		//Wait for Delay, copy Data and then next step
		IF NOT fbMBRead_FC3.bBusy AND NOT fbMBRead_FC3.bError AND timer_Delay.Q THEN
			m_Poll_ok:=TRUE;
			int_Data_Received:=int_Data_Received+1;
			m_MBTCPError := FALSE; 
			
			FOR i:=0 TO 9 BY 1 DO
				arrBuffer_Received[i + WORD_TO_INT(w_Adress)] := arrBuffer_FC3[i];
			END_FOR
			
			//Go to Next Step
			timer_Timeout.IN := FALSE;
			fbMBRead_FC3.bExecute := FALSE;
			timer_Delay.IN := FALSE;		
			iStateModbusRead := iStateModbusRead+1;
		END_IF	

		//Error or Timeout
		IF FPError_FC_3.Q THEN 
			iStateModbusError := 300;
			int_FC4Error := int_FC4Error+1;
		ELSIF timer_Timeout.Q THEN  
			timer_Timeout.IN := FALSE; 	
			iStateModbusError := 300;
			int_TimeoutError := int_TimeoutError+1;
		END_IF
	
	9://Wait and go to next step
		timer_Wait.IN := TRUE;
		
		IF timer_Wait.Q = TRUE THEN
			iStateModbusRead := iStateModbusRead+1;
			timer_Wait.IN :=FALSE;
		END_IF
		
	10: // clean the array  Poll 4
		FOR i:=0 TO 10 BY 1 DO
			arrBuffer_FC3[i] := 0;
		END_FOR
		w_Adress := w_Adress + 10;
		usint_Quantity := 10; 
		iStateModbusRead := iStateModbusRead+1;
		
	11://read the required registers
		//Start Read Poll 4
		fbMBRead_FC3.nQuantity := usint_Quantity;
		fbMBRead_FC3.nMBAddr := w_Adress;
		fbMBRead_FC3.bExecute := TRUE;
		fbMBRead_FC3.nUnitID := 1;
		timer_Timeout.IN := TRUE;
		IF fbMBRead_FC3.bBusy THEN 
			timer_Delay.IN := TRUE; 
		END_IF
		
		//Wait for Delay, copy Data and then next step
		IF NOT fbMBRead_FC3.bBusy AND NOT fbMBRead_FC3.bError AND timer_Delay.Q THEN
			m_Poll_ok:=TRUE;
			int_Data_Received:=int_Data_Received+1;
			m_MBTCPError := FALSE; 
			
			FOR i:=0 TO 9 BY 1 DO
				arrBuffer_Received[i + WORD_TO_INT(w_Adress)] := arrBuffer_FC3[i];
			END_FOR
			
			//Go to Next Step
			timer_Timeout.IN := FALSE;
			fbMBRead_FC3.bExecute := FALSE;
			timer_Delay.IN := FALSE;		
			iStateModbusRead := iStateModbusRead+1;
		END_IF	

		//Error or Timeout
		IF FPError_FC_3.Q THEN 
			iStateModbusError := 300;
			int_FC4Error := int_FC4Error+1;
		ELSIF timer_Timeout.Q THEN  
			timer_Timeout.IN := FALSE; 	
			iStateModbusError := 300;
			int_TimeoutError := int_TimeoutError+1;
		END_IF
	
	12://Wait and go to next step
		timer_Wait.IN := TRUE;
		
		IF timer_Wait.Q = TRUE THEN
			iStateModbusRead := iStateModbusRead+1;
			timer_Wait.IN :=FALSE;
		END_IF		
		
	13: // clean the array  Poll 4
		FOR i:=0 TO 10 BY 1 DO
			arrBuffer_FC3[i] := 0;
		END_FOR
		w_Adress := w_Adress + 10;
		usint_Quantity := 10; 
		iStateModbusRead := iStateModbusRead+1;
		
	14://read the required registers
		//Start Read Poll 4
		fbMBRead_FC3.nQuantity := usint_Quantity;
		fbMBRead_FC3.nMBAddr := w_Adress;
		fbMBRead_FC3.bExecute := TRUE;
		fbMBRead_FC3.nUnitID := 1;
		timer_Timeout.IN := TRUE;
		IF fbMBRead_FC3.bBusy THEN 
			timer_Delay.IN := TRUE; 
		END_IF
		
		//Wait for Delay, copy Data and then next step
		IF NOT fbMBRead_FC3.bBusy AND NOT fbMBRead_FC3.bError AND timer_Delay.Q THEN
			m_Poll_ok:=TRUE;
			int_Data_Received:=int_Data_Received+1;
			m_MBTCPError := FALSE; 
			
			FOR i:=0 TO 9 BY 1 DO
				arrBuffer_Received[i + WORD_TO_INT(w_Adress)] := arrBuffer_FC3[i];
			END_FOR
			
			//Go to Next Step
			timer_Timeout.IN := FALSE;
			fbMBRead_FC3.bExecute := FALSE;
			timer_Delay.IN := FALSE;		
			iStateModbusRead := iStateModbusRead+1;
		END_IF	

		//Error or Timeout
		IF FPError_FC_3.Q THEN 
			iStateModbusError := 300;
			int_FC4Error := int_FC4Error+1;
		ELSIF timer_Timeout.Q THEN  
			timer_Timeout.IN := FALSE; 	
			iStateModbusError := 300;
			int_TimeoutError := int_TimeoutError+1;
		END_IF
	
	15://Wait and go to next step
		timer_Wait.IN := TRUE;
		
		IF timer_Wait.Q = TRUE THEN
			iStateModbusRead := iStateModbusRead+1;
			timer_Wait.IN :=FALSE;
		END_IF
		
	16: // clean the array  Poll 5
		FOR i:=0 TO 10 BY 1 DO
			arrBuffer_FC3[i] := 0;
		END_FOR
		w_Adress := w_Adress + 10;
		usint_Quantity := 10; 
		iStateModbusRead := iStateModbusRead+1;
		
	17://read the required registers
		//Start Read Poll 5
		fbMBRead_FC3.nQuantity := usint_Quantity;
		fbMBRead_FC3.nMBAddr := w_Adress;
		fbMBRead_FC3.bExecute := TRUE;
		fbMBRead_FC3.nUnitID := 1;
		timer_Timeout.IN := TRUE;
		IF fbMBRead_FC3.bBusy THEN 
			timer_Delay.IN := TRUE; 
		END_IF
		
		//Wait for Delay, copy Data and then next step
		IF NOT fbMBRead_FC3.bBusy AND NOT fbMBRead_FC3.bError AND timer_Delay.Q THEN
			m_Poll_ok:=TRUE;
			int_Data_Received:=int_Data_Received+1;
			m_MBTCPError := FALSE; 
			
			FOR i:=0 TO 9 BY 1 DO
				arrBuffer_Received[i + WORD_TO_INT(w_Adress)] := arrBuffer_FC3[i];
			END_FOR
			
			//Go to Next Step
			timer_Timeout.IN := FALSE;
			fbMBRead_FC3.bExecute := FALSE;
			timer_Delay.IN := FALSE;		
			iStateModbusRead := iStateModbusRead+1;
		END_IF	

		//Error or Timeout
		IF FPError_FC_3.Q THEN 
			iStateModbusError := 300;
			int_FC4Error := int_FC4Error+1;
		ELSIF timer_Timeout.Q THEN  
			timer_Timeout.IN := FALSE; 	
			iStateModbusError := 300;
			int_TimeoutError := int_TimeoutError+1;
		END_IF
	
	18://Wait and go to next step
		timer_Wait.IN := TRUE;
		
		IF timer_Wait.Q = TRUE THEN
			iStateModbusRead := iStateModbusRead+1;
			timer_Wait.IN :=FALSE;
		END_IF	

	19: // clean the array  Poll 6
		FOR i:=0 TO 10 BY 1 DO
			arrBuffer_FC3[i] := 0;
		END_FOR
		w_Adress := w_Adress + 10;
		usint_Quantity := 10; 
		iStateModbusRead := iStateModbusRead+1;
		
	20://read the required registers
		//Start Read Poll 6
		fbMBRead_FC3.nQuantity := usint_Quantity;
		fbMBRead_FC3.nMBAddr := w_Adress;
		fbMBRead_FC3.bExecute := TRUE;
		fbMBRead_FC3.nUnitID := 1;
		timer_Timeout.IN := TRUE;
		IF fbMBRead_FC3.bBusy THEN 
			timer_Delay.IN := TRUE; 
		END_IF
		
		//Wait for Delay, copy Data and then next step
		IF NOT fbMBRead_FC3.bBusy AND NOT fbMBRead_FC3.bError AND timer_Delay.Q THEN
			m_Poll_ok:=TRUE;
			int_Data_Received:=int_Data_Received+1;
			m_MBTCPError := FALSE; 
			
			FOR i:=0 TO 9 BY 1 DO
				arrBuffer_Received[i + WORD_TO_INT(w_Adress)] := arrBuffer_FC3[i];
			END_FOR
			
			//Go to Next Step
			timer_Timeout.IN := FALSE;
			fbMBRead_FC3.bExecute := FALSE;
			timer_Delay.IN := FALSE;		
			iStateModbusRead := iStateModbusRead+1;
		END_IF	

		//Error or Timeout
		IF FPError_FC_3.Q THEN 
			iStateModbusError := 300;
			int_FC4Error := int_FC4Error+1;
		ELSIF timer_Timeout.Q THEN  
			timer_Timeout.IN := FALSE; 	
			iStateModbusError := 300;
			int_TimeoutError := int_TimeoutError+1;
		END_IF
	
	21://Wait and go to next step
		timer_Wait.IN := TRUE;
		
		IF timer_Wait.Q = TRUE THEN
			iStateModbusRead := iStateModbusRead+1;
			timer_Wait.IN :=FALSE;
		END_IF	
		
	22: // clean the array  Poll 7
		FOR i:=0 TO 10 BY 1 DO
			arrBuffer_FC3[i] := 0;
		END_FOR
		w_Adress := w_Adress + 10;
		usint_Quantity := 10; 
		iStateModbusRead := iStateModbusRead+1;
		
	23://read the required registers
		//Start Read Poll 7
		fbMBRead_FC3.nQuantity := usint_Quantity;
		fbMBRead_FC3.nMBAddr := w_Adress;
		fbMBRead_FC3.bExecute := TRUE;
		fbMBRead_FC3.nUnitID := 1;
		timer_Timeout.IN := TRUE;
		IF fbMBRead_FC3.bBusy THEN 
			timer_Delay.IN := TRUE; 
		END_IF
		
		//Wait for Delay, copy Data and then next step
		IF NOT fbMBRead_FC3.bBusy AND NOT fbMBRead_FC3.bError AND timer_Delay.Q THEN
			m_Poll_ok:=TRUE;
			int_Data_Received:=int_Data_Received+1;
			m_MBTCPError := FALSE; 
			
			FOR i:=0 TO 9 BY 1 DO
				arrBuffer_Received[i + WORD_TO_INT(w_Adress)] := arrBuffer_FC3[i];
			END_FOR
			
			//Go to Next Step
			timer_Timeout.IN := FALSE;
			fbMBRead_FC3.bExecute := FALSE;
			timer_Delay.IN := FALSE;		
			iStateModbusRead := iStateModbusRead+1;
		END_IF	

		//Error or Timeout
		IF FPError_FC_3.Q THEN 
			iStateModbusError := 300;
			int_FC4Error := int_FC4Error+1;
		ELSIF timer_Timeout.Q THEN  
			timer_Timeout.IN := FALSE; 	
			iStateModbusError := 300;
			int_TimeoutError := int_TimeoutError+1;
		END_IF
	
	24://Wait and go to next step
		timer_Wait.IN := TRUE;
		
		IF timer_Wait.Q = TRUE THEN
			iStateModbusRead := iStateModbusRead+1;
			timer_Wait.IN :=FALSE;
		END_IF	

	25: // clean the array  Poll 8
		FOR i:=0 TO 10 BY 1 DO
			arrBuffer_FC3[i] := 0;
		END_FOR
		w_Adress := w_Adress + 10;
		usint_Quantity := 2;		// only 2 possible, otherwise out of the range 
		iStateModbusRead := iStateModbusRead+1;
		
	26://read the required registers
		//Start Read Poll 8
		fbMBRead_FC3.nQuantity := usint_Quantity;
		fbMBRead_FC3.nMBAddr := w_Adress;
		fbMBRead_FC3.bExecute := TRUE;
		fbMBRead_FC3.nUnitID := 1;
		timer_Timeout.IN := TRUE;
		IF fbMBRead_FC3.bBusy THEN 
			timer_Delay.IN := TRUE; 
		END_IF
		
		//Wait for Delay, copy Data and then next step
		IF NOT fbMBRead_FC3.bBusy AND NOT fbMBRead_FC3.bError AND timer_Delay.Q THEN
			m_Poll_ok:=TRUE;
			int_Data_Received:=int_Data_Received+1;
			m_MBTCPError := FALSE; 
			
			FOR i:=0 TO 9 BY 1 DO
				arrBuffer_Received[i + WORD_TO_INT(w_Adress)] := arrBuffer_FC3[i];
			END_FOR
			
			//Go to Next Step
			timer_Timeout.IN := FALSE;
			fbMBRead_FC3.bExecute := FALSE;
			timer_Delay.IN := FALSE;		
			iStateModbusRead := 30;  // convert data
		END_IF	

		//Error or Timeout
		IF FPError_FC_3.Q THEN 
			iStateModbusError := 300;
			int_FC4Error := int_FC4Error+1;
		ELSIF timer_Timeout.Q THEN  
			timer_Timeout.IN := FALSE; 	
			iStateModbusError := 300;
			int_TimeoutError := int_TimeoutError+1;
		END_IF
	

	
	30: // convert data
		real_VoltageL1N_V	:= DINT_TO_REAL((DWORD_TO_DINT(arrBuffer_Received[13] * 65536 + arrBuffer_Received[12]))) /1000;

		real_VoltageL1N_V 	:= WORD_TO_REAL(arrBuffer_Received[0]) /10;
		real_VoltageL2N_V 	:= WORD_TO_REAL(arrBuffer_Received[2]) /10;
		real_VoltageL3N_V 	:= WORD_TO_REAL(arrBuffer_Received[4]) /10;
		real_VoltageL1L2_V 	:= WORD_TO_REAL(arrBuffer_Received[6]) /10;
		real_VoltageL2L3_V 	:= WORD_TO_REAL(arrBuffer_Received[8]) /10;
		real_VoltageL3L1_V 	:= WORD_TO_REAL(arrBuffer_Received[10]) /10;


		real_CurrentL1_A	:= DINT_TO_REAL((DWORD_TO_DINT(arrBuffer_Received[13] * 65536 + arrBuffer_Received[12]))) /1000;
		real_CurrentL2_A	:= DINT_TO_REAL((DWORD_TO_DINT(arrBuffer_Received[15] * 65536 + arrBuffer_Received[14]))) /1000;
		real_CurrentL3_A	:= DINT_TO_REAL((DWORD_TO_DINT(arrBuffer_Received[17] * 65536 + arrBuffer_Received[16]))) /1000;	
		
		real_RealPowerL1_kW	:= DINT_TO_REAL((DWORD_TO_DINT(arrBuffer_Received[19] * 65536 + arrBuffer_Received[18]))) /10000;
		real_RealPowerL2_kW	:= DINT_TO_REAL((DWORD_TO_DINT(arrBuffer_Received[21] * 65536 + arrBuffer_Received[20]))) /10000;
		real_RealPowerL3_kW	:= DINT_TO_REAL((DWORD_TO_DINT(arrBuffer_Received[23] * 65536 + arrBuffer_Received[22]))) /10000;	

		real_RealPower_kW	:= DINT_TO_REAL((DWORD_TO_DINT(arrBuffer_Received[41] * 65536 + arrBuffer_Received[40]))) /10000;

		real_ApparentPower_kVA	:= DINT_TO_REAL((DWORD_TO_DINT(arrBuffer_Received[43] * 65536 + arrBuffer_Received[42]))) /10000;
		real_ReactivePower_kVAr	:= DINT_TO_REAL((DWORD_TO_DINT(arrBuffer_Received[45] * 65536 + arrBuffer_Received[44]))) /10000;

		real_Frequency_Hz	:= WORD_TO_REAL(arrBuffer_Received[51]) /10;


		real_EnergyTotal_Import_kWh		:= DINT_TO_REAL((DWORD_TO_DINT(arrBuffer_Received[53] * 65536 + arrBuffer_Received[52]))) /10;
		real_EnergyTotal_Export_kWh		:= DINT_TO_REAL((DWORD_TO_DINT(arrBuffer_Received[79] * 65536 + arrBuffer_Received[78]))) /10;
		real_EnergyTotal_ExportT1_kWh	:= DINT_TO_REAL((DWORD_TO_DINT(arrBuffer_Received[71] * 65536 + arrBuffer_Received[70]))) /10;
		real_EnergyTotal_ExportT2_kWh	:= DINT_TO_REAL((DWORD_TO_DINT(arrBuffer_Received[73] * 65536 + arrBuffer_Received[72]))) /10;
		real_EnergyTotal_ExportT3_kWh	:= DINT_TO_REAL((DWORD_TO_DINT(arrBuffer_Received[75] * 65536 + arrBuffer_Received[74]))) /10;
		real_EnergyTotal_ExportT4_kWh	:= DINT_TO_REAL((DWORD_TO_DINT(arrBuffer_Received[77] * 65536 + arrBuffer_Received[76]))) /10;
		
		// go to next state
		iStateModbusRead := iStateModbusRead+1;		
		
	31://Wait and go to start
		timer_Wait.IN := TRUE;
		
		IF timer_Wait.Q = TRUE THEN
			iStateModbusRead := 1;
			timer_Wait.IN :=FALSE;
		END_IF	

END_CASE

(* wait timer*)

timer_Wait(PT:=T#1S);


(*------------------------------------------------------------------Error and Warning----------------------------------------------------------------------------*)	
 
timer_Connection_ok			(In:=int_Data_Received<>int_Data_Received_old,PT:=T#10S);
timer_Connection_ok_TOF		(In:=NOT(int_Data_Received<>int_Data_Received_old) AND int_Data_Received>3 ,PT:=T#20S);
int_Data_Received_old:=int_Data_Received;
m_PollSuccessful:=NOT timer_Connection_ok.Q AND timer_Connection_ok_TOF.Q ;

(*------------------------------------------------------------------------------------------Modbus TCP Functions---------------------------------------------------------------------------------------------*)

fbMBRead_FC3(	sIPAddr:= str_IPAdress, 
				nTCPPort:= 502,
				cbLength:= SIZEOF(arrBuffer_FC3), 
				pDestAddr:= ADR(arrBuffer_FC3), 
				tTimeout:= T#10S,
				nErrId => udint_Error_ID);

FPError_FC_3(CLK:= fbMBRead_FC3.bError, Q=> );		

(*------------------------------------------------------------------------------------------State Machine Error---------------------------------------------------------------------------------------------*)	

CASE iStateModbusError OF
	
	300://Error
		timer_Wait.IN :=TRUE;
		timer_Delay.IN := FALSE;
		fbMBRead_FC3.bExecute := FALSE;
		m_MBTCPError := TRUE; 		
		m_Poll_ok:=FALSE;
		int_Data_Received:=0;
		
				//Restart from new with the Read out part after an Error
		IF timer_Wait.Q = TRUE THEN
			iStateModbusRead := 0;	
			iStateModbusError := 0;
			timer_Wait.IN :=FALSE;
			timer_Timeout.IN := FALSE;
		END_IF		
							
END_CASE

END_FUNCTION_BLOCK

// ---- FBs/CTA/Optiplus3/FB_HP_CTA_Optiplus3_Modular.TcPOU
FUNCTION_BLOCK FB_HP_CTA_Optiplus3_Modular
VAR_INPUT PERSISTENT
	bEnable									: BOOL;												//{#lynus.ag#()} //Enable the Fuctionblock and his logic
	bPowerDataInvers						: BOOL;												//With True its possible to invert all received power data from the electric meter
	byUnitID								: BYTE;												//Unit ID fromt the Soltop M-Tec Modbus Server(0 to 255)
	diNrOfEMS_IN							: DINT;												//Number of EMS what control this Device.
	diNrOfEM_IN_HP							: DINT;												//Number of the electric meter for incoming power data. (Power Data for this Device)
	sIPAdress								: STRING(15);										//IP Adress from the oltop M-Tec Modbus Server
	stSetupHP								: ST_Setup_HP;										//{#lynus.ag#()} //Setup heating pump
END_VAR
VAR_INPUT
END_VAR
VAR_OUTPUT
	stDataHP								: ST_HP_Output;										//{#lynus.ag#()} //Output Data Heating pump
	stDataTempS								: ST_Temperature_Output;							//Temperature output data
	diNrOfHP_OUT							: DINT;												//Active Number from the heating pump for using on other functions		
	diNrOfTempS_OUT_ServiceWaterTop			: DINT;												//Active Number from the Temperature Sensor for using on other functions
END_VAR
VAR
	{attribute 'hide'}
	fbHP									: FB_HeatingPump;									//Function block for heating pump
	{attribute 'hide'}
	fbNumberDevice							: FB_NumberOfDevice;								//Function block to calcualte the number of the Device
	{attribute 'hide'}
	fbNumberDevice_Temp						: FB_NumberOfDevice;								//Function block to calcualte the number of the Device
	{attribute 'hide'}
	fbConvertWordToDword					: FB_CV_WORD_TO_DWORD;								//Convert function
	{attribute 'hide'}
	fbConvertDwordToWord					: FB_CV_DWORD_TO_WORD;								//Convert function
	{attribute 'hide'}
	fbTempS									: FB_TempSensor_M50_P200;							//Function for Temperature Sensor
	fbDIExternalLock						: FB_XL1XXX_DI;										//Digital Input from external loock signal
	{attribute 'hide'}
	timDissableFunctions					: TON;												//Timer to dissable the Function after Lynus_Standards.Constants_General.tTimeDissableLynusFunctions Days without connection to the Lynus Cloud
	{attribute 'hide'}
	timResetConnectionOnGVL					: TON;												//Timer to try reset the connection Flag on the GVL. (When somebody delete the Connection Function and make only a onlinechange)
	{attribute 'hide'}
	timGetTime								: TON;												//Timer to activate the function tho read out the windows system time
	{attribute 'hide'}
	timDelay								: TON;												//Timer for Delay between Requests
	{attribute 'hide'}
	timTimeout								: TON;												//Timer for Timeout
	{attribute 'hide'}
	FNReset									: F_TRIG;											//Internal negative edge
	{attribute 'hide'}
	FPEnable								: R_TRIG;											//Internal positive Edge
	{attribute 'hide'}
	FNTimDissable							: F_TRIG;											//Internal negative Edge
	{attribute 'hide'}
	FPError_FC_4							: R_TRIG;											//Internal positive Edge
	{attribute 'hide'}
	FPError_FC_16							: R_TRIG;											//Internal positive Edge
	{attribute 'hide'}
	fbGetSystemTime							: NT_GetTime;										//Function to read out the windows system time on the local plc
	{attribute 'hide'}
	arrPD									: ARRAY[1..21] OF FB_PersistentData_Number;			//Function to save persistent data
	{attribute 'hide'}
	fbPDString								: FB_PersistentData_String;							//Function to save persistent string data
	{attribute 'hide'}
	fbMBRead_FC4							: FB_MBReadInputRegs ;								//Modbus Read Function (FC4)
	{attribute 'hide'}
	fbMBWrite_FC16							: FB_MBWriteRegs ;									//Modbus Write Function (FC16)
	{attribute 'hide'}
	stFloat									: ST_UN_FLOAT_CONVERT_DWORD_REAL;					//Convert the Float Raw Value
	{attribute 'hide'}
	arrCounterForGVL						: ARRAY[1..2] OF DINT;								//Counter to clean old data on GVL
	{attribute 'hide'}
	arrBuffer_FC4							: ARRAY[1..16] OF WORD;								//Buffer with Data from FC4
	{attribute 'hide'}
	arrBuffer_FC16							: ARRAY[1..8] OF WORD;								//Buffer with Data from FC16
	{attribute 'hide'}
	arrAlarmList							: ARRAY[1..6] OF DINT;								//Array with the Alarm List from the Heating pump
	{attribute 'hide'}
	arrHPState								: ARRAY[1..2] OF REAL;								//Heating pump actual State to say that the pump is running or not
	{attribute 'hide'}
	bGroupErrorHP							: BOOL;												//Group Error from the Heating Pump
	{attribute 'hide'}
	bHPIsRunning							: BOOL;												//Feedback from the HP if its running or not
	{attribute 'hide'}
	bErrorTempSensorBoilerServiceWaterTop	: BOOL;												//Error for the Temp Senor top in the service water boiler
	{attribute 'hide'}
	bMBTCPError								: BOOL;												//Modbus TCP Error
	{attribute 'hide'}
	byWaitInStep							: BYTE;												//Wait in Step before start to clean data on PLC
	{attribute 'hide'}
	iStateGVLData							: INT;												//State machine to handle the data on the GVL
	{attribute 'hide'}
	iStateModbusRead						: INT;												//State variable for Statemachine
	{attribute 'hide'}
	iStateModbusWrite						: INT;												//State variable for Statemachine
	{attribute 'hide'}
	iStateModbusError						: INT;												//State variable for Statemachine
	{attribute 'hide'}
	iStateModbus_CP							: INT;												//Compare State variable
	{attribute 'hide'}
	rTB4									: REAL;												//Temp. Sensor Top in the Heating Boiler
	{attribute 'hide'}
	rTB41									: REAL;												//Temp. Sensor Below in the Heating Boiler
	{attribute 'hide'}
	diNumberOfActiveBatterys				: DINT;												//Number of active batterys
	{attribute 'hide'}
	diNumberOfBatteryInverterInEPO			: DINT;												//Number of battery inverters that work in Emergency Power operation 
	{attribute 'hide'}
	diLPForGVL								: DINT;												//Loop to clean old data on GVL
	{attribute 'hide'}	
	dwSumSOC								: DWORD;											//Sum of the SOC from all batterys
	{attribute 'hide'}
	rNewPowerToHP							: REAL;												//New surplus power fpr the HP in W
	{attribute 'hide'}
	lrGridPower								: LREAL;											//Grid power in kW
	{attribute 'hide'}
	lrSizeGridConnection					: LREAL;											//Size of the complete grid connection
	{attribute 'hide'}
	liLPBatteryData							: LINT;												//Loop to check some data from batterys
	{attribute 'hide'}
	liLPInEPO								: LINT;												//Loop to check if 1 or more battery inverters build a island grid	
	{attribute 'hide'}
	liLPGridData							: LINT;												//Loop to check some grid data
END_VAR
VAR PERSISTENT
	{attribute 'conditionalshow'}
	diNrOfEMS_IN_CP							: DINT;												//Number of EMS what control this Device to compare with the original
END_VAR

//Creator : Kai Ebensperger
//Company : Lynus AG
//Date : 15.02.2022
//Version : 1.0.0.0

//With this function block its possible to control a Heating pump from the Factory CTA
//The communication is over Modbus TCP.
//The Device on the Soltop side is called Optiplus 3.
//The excess power can be transferred to this pump linearly as it is modulating. The power can be transferred in watts.
//Versions that are supported : V1.10.1
//This Heating pump can by control with a surplus on PV Power in Watt. This power can send directly to the Heating Pump and the Heating pump uses it where it is needed or it can be consumed.

//NOTE for diNr.....Designation => 
//_IN = Here Data come in from other Functions or go out to other functions about the GVL
//_OUT = Here Data go out to other functions about the GVL

(*------------------------------------------------------------Limits----------------------------------------------------------------------------------*)

diNrOfEMS_IN := LIMIT(0,diNrOfEMS_IN,Constants_Energy.diMaxNumberOfEMS);
	diNrOfEM_IN_HP := LIMIT(0,diNrOfEM_IN_HP,Constants_Energy.diMaxNumberOfElectricMeters);
			
(*------------------------------------------------------------------Power Data----------------------------------------------------------------------------*)

IF NOT bPowerDataInvers THEN
	fbHP.lrCounterEnergyT1_Consumption := Lynus_Standards.GVL_Energy.stDataElectricMeters[diNrOfEM_IN_HP].lrCounterEnergyT1_Production * 1000;
	fbHP.lrCounterEnergyT2_Consumption := Lynus_Standards.GVL_Energy.stDataElectricMeters[diNrOfEM_IN_HP].lrCounterEnergyT2_Production * 1000;
	fbHP.lrCounterEnergyT1_Production := Lynus_Standards.GVL_Energy.stDataElectricMeters[diNrOfEM_IN_HP].lrCounterEnergyT1_Consumption * 1000;
	fbHP.lrCounterEnergyT2_Production := Lynus_Standards.GVL_Energy.stDataElectricMeters[diNrOfEM_IN_HP].lrCounterEnergyT1_Consumption * 1000;
	fbHP.lrTotalCounterEnergy_Consumption := Lynus_Standards.GVL_Energy.stDataElectricMeters[diNrOfEM_IN_HP].lrTotalCounterEnergy_Production * 1000;
	fbHP.lrTotalCounterEnergy_Production := Lynus_Standards.GVL_Energy.stDataElectricMeters[diNrOfEM_IN_HP].lrTotalCounterEnergy_Consumption * 1000;
		fbHP.lrElPowerHP := (Lynus_Standards.GVL_Energy.stDataElectricMeters[diNrOfEM_IN_HP].lrPower * 1000) * - 1;
ELSE
	fbHP.lrCounterEnergyT1_Consumption := Lynus_Standards.GVL_Energy.stDataElectricMeters[diNrOfEM_IN_HP].lrCounterEnergyT1_Consumption * 1000;
	fbHP.lrCounterEnergyT2_Consumption := Lynus_Standards.GVL_Energy.stDataElectricMeters[diNrOfEM_IN_HP].lrCounterEnergyT2_Consumption * 1000;
	fbHP.lrCounterEnergyT1_Production := Lynus_Standards.GVL_Energy.stDataElectricMeters[diNrOfEM_IN_HP].lrCounterEnergyT1_Production * 1000;
	fbHP.lrCounterEnergyT2_Production := Lynus_Standards.GVL_Energy.stDataElectricMeters[diNrOfEM_IN_HP].lrCounterEnergyT2_Production * 1000;
	fbHP.lrTotalCounterEnergy_Consumption := Lynus_Standards.GVL_Energy.stDataElectricMeters[diNrOfEM_IN_HP].lrTotalCounterEnergy_Consumption * 1000;
	fbHP.lrTotalCounterEnergy_Production := Lynus_Standards.GVL_Energy.stDataElectricMeters[diNrOfEM_IN_HP].lrTotalCounterEnergy_Production * 1000;
		fbHP.lrElPowerHP := Lynus_Standards.GVL_Energy.stDataElectricMeters[diNrOfEM_IN_HP].lrPower * 1000;
END_IF

(*-------------------------------------------------------------Calcualte the number of HP and Temperature---------------------------------------------------------------*)

fbNumberDevice(
	diActualNumberOfDevices:= Lynus_Standards.GVL_Energy.stNumberOfDevices.diNumberOfHP, 
	diMaxNumberOfDevices:= Constants_Energy.diMaxNumberOfHeatingPumps, 
	udiCounterOnlineChange:= TwinCAT_SystemInfoVarList._AppInfo.OnlineChangeCnt, 
	bNumberIsCalculatet=> , 
	bFPNumberIsCalculatet=> , 
	bOnlineChange=> , 
	diNumberForThisDevice=> diNrOfHP_OUT, 
	diNumberOfTotalDevices=> );

//Write new Numer on GVL
IF fbNumberDevice.bFPNumberIsCalculatet THEN
	Lynus_Standards.GVL_Energy.stNumberOfDevices.diNumberOfHP := fbNumberDevice.diNumberOfTotalDevices;	
END_IF 

//Delete old Number on GVL
IF fbNumberDevice.bOnlineChange THEN 
	Lynus_Standards.GVL_Energy.stNumberOfDevices.diNumberOfHP := diNrOfHP_OUT;	
		iStateGVLData := 1; 
END_IF
	
fbNumberDevice_Temp(
	diActualNumberOfDevices:= Lynus_Standards.GVL_Sensors.diNumberOfTemperatureSensors, 
	diMaxNumberOfDevices:= Constants_Sensors.diMaxNumberOfTemperatureSensors, 
	udiCounterOnlineChange:= TwinCAT_SystemInfoVarList._AppInfo.OnlineChangeCnt, 
	bNumberIsCalculatet=> , 
	bFPNumberIsCalculatet=> , 
	bOnlineChange=> , 
	diNumberForThisDevice=> diNrOfTempS_OUT_ServiceWaterTop, 
	diNumberOfTotalDevices=> );	

//Write new Numer on GVL
IF fbNumberDevice_Temp.bFPNumberIsCalculatet THEN
	Lynus_Standards.GVL_Sensors.diNumberOfTemperatureSensors := fbNumberDevice.diNumberOfTotalDevices;	
END_IF 

//Delete old Number on GVL
IF fbNumberDevice_Temp.bOnlineChange THEN 
	Lynus_Standards.GVL_Sensors.diNumberOfTemperatureSensors := diNrOfTempS_OUT_ServiceWaterTop;	
		iStateGVLData := 1; 
END_IF

(*-------------------------------------------------------------Get the local windows system time for this plc---------------------------------------------------------------*)
timGetTime(IN:= bEnable AND NOT timGetTime.Q, PT:= T#30S, Q=> , ET=> );

fbGetSystemTime(
	NETID:= , 
	START:= timGetTime.Q AND NOT fbGetSystemTime.BUSY, 
	TMOUT:= , 
	BUSY=> , 
	ERR=> , 
	ERRID=> , 
	TIMESTR=> );	

fbHP.stSystemTime.wHour := fbGetSystemTime.TIMESTR.wHour;
	fbHP.stSystemTime.wMinute := fbGetSystemTime.TIMESTR.wMinute;	

(*-------------------------------------------------------------Service from Backend is ready and check the connection to backen for dissabel/enable Function---------------------------------------------------------------*)

//Try to reset the variable for connection on the GVL. When all is normal then the Lynus Mqtt connection function set this variable to true in the next cycle
//When we have no connection to the backend then after Lynus_Standards.Constants_General.tTimeDissableLynusFunctions days the Function is dissabled with all of his functionalities
timResetConnectionOnGVL(IN:= NOT timResetConnectionOnGVL.Q, PT:= T#1H, Q=> , ET=> );
	IF timResetConnectionOnGVL.Q THEN Lynus_Standards.GVL_Communicator.bStateConnectionToEnableFunctions := FALSE; END_IF
		IF NOT Lynus_Standards.GVL_Communicator.bStateConnectionToEnableFunctions THEN timDissableFunctions.IN := TRUE; ELSE timDissableFunctions.IN := FALSE; END_IF  
			timDissableFunctions(IN:= , PT:= Lynus_Standards.Constants_General.tTimeDissableLynusFunctions, Q=> , ET=> );		
	
(*------------------------------------------------------------------Logic----------------------------------------------------------------------------*)

//Calcualte the total SOC if we have more then 1 battery in our system
diNumberOfActiveBatterys := 0;
	dwSumSOC := 0;
		FOR liLPBatteryData := 1 TO Constants_Energy.diMaxNumberOfBatterys BY 1 DO
			IF Lynus_Standards.GVL_Energy.stDataOfBatterys[diNrOfEMS_IN,liLPBatteryData].bEnabled THEN diNumberOfActiveBatterys := diNumberOfActiveBatterys + 1; END_IF
				dwSumSOC := dwSumSOC + Lynus_Standards.GVL_Energy.stDataOfBatterys[diNrOfEMS_IN,liLPBatteryData].dwSOC;
		END_FOR
	
IF diNumberOfActiveBatterys > 0 THEN
	fbHP.dwBatterySOC := DINT_TO_DWORD(DWORD_TO_DINT(dwSumSOC) / diNumberOfActiveBatterys);
ELSE
	fbHP.dwBatterySOC := 100;	//When we have no battery in the ems system
END_IF

//Check if one or more Batterysystems or batteryinverter make island mode
diNumberOfBatteryInverterInEPO := 0;
	FOR liLPInEPO := 1 TO Constants_Energy.diMaxNumberOfBatteryInverters BY 1 DO
		IF Lynus_Standards.GVL_Energy.stDataOfBatteryInverters[diNrOfEMS_IN,liLPInEPO].bWorkOnIslandMode THEN fbHP.bEPOIsActive := TRUE; diNumberOfBatteryInverterInEPO := diNumberOfBatteryInverterInEPO + 1; END_IF
	END_FOR 
		IF diNumberOfBatteryInverterInEPO <= 0 THEN fbHP.bEPOIsActive := FALSE; END_IF

//Check the max. power of the grid connection and the sum of grid power
lrSizeGridConnection := 0;
	lrGridPower := 0;
		FOR liLPGridData := 1 TO Constants_Energy.diMaxNumberOfGridConnections BY 1 DO
			lrSizeGridConnection := lrSizeGridConnection + Lynus_Standards.GVL_Energy.stDataGridConnections[diNrOfEMS_IN,liLPGridData].rSizeGridConn;
				lrGridPower := lrGridPower + Lynus_Standards.GVL_Energy.stDataGridConnections[diNrOfEMS_IN,liLPGridData].lrPower;
		END_FOR		

//Set the target power from the EMS to the HP Function
fbHP.arrTargetPower[1] := Lynus_Standards.GVL_Energy.stDataHeatingPumps[diNrOfEMS_IN,diNrOfHP_OUT].arrTargetPowerEMS[1];

	stSetupHP.rMaxPower2 := 0;
		fbHP.arrTargetPower[2] := 0;
		
//Digital input for external lock signal
fbDIExternalLock(bInvers:= FALSE, bSignal=> );

(*------------------------------------------------------------------------------------------State Machine Read---------------------------------------------------------------------------------------------*)

//Start the Statemachine
FPEnable(CLK:= bEnable, Q=> );
	FNTimDissable(CLK:= timDissableFunctions.Q, Q=> );
		IF (FPEnable.Q AND iStateModbusRead = 0 AND iStateModbusRead = 0 AND iStateModbusError = 0) OR
			(bEnable AND FNTimDissable.Q AND iStateModbusRead = 0 AND iStateModbusRead = 0 AND iStateModbusError = 0) THEN 
				iStateModbusRead := 1; 
		END_IF
			IF NOT bEnable THEN iStateModbusRead := 0; iStateModbusWrite := 0; iStateModbusError := 0; END_IF

//Timer for delay
timDelay(IN:= , PT:= T#250MS, Q=> , ET=> );	

//Timer for Timeout in Statemachine
IF (iStateModbusRead > 0 AND iStateModbusRead <= 4 AND iStateModbusRead = iStateModbus_CP) OR
		(iStateModbusWrite > 0 AND iStateModbusWrite <= 2 AND iStateModbusWrite = iStateModbus_CP) THEN
			timTimeout.IN := TRUE;
ELSE	
			timTimeout.IN := FALSE;
END_IF 
	IF iStateModbusRead = 0 AND iStateModbusWrite = 0 THEN timTimeout.IN := FALSE; END_IF
		timTimeout(IN:= , PT:= T#20S, Q=> , ET=> );
	
CASE iStateModbusRead OF
	
	0://Init
		iStateModbus_CP := 0;
			timDelay.IN := FALSE;
			
		fbMBWrite_FC16.bExecute := FALSE;
			fbMBRead_FC4.bExecute := FALSE;
				bHPIsRunning := FALSE;
					rTB4 := 0;
						rTB41 := 0;	
							arrAlarmList[1] := 0; arrAlarmList[2] := 0; arrAlarmList[3] := 0; arrAlarmList[4] := 0; arrAlarmList[5] := 0; arrAlarmList[6] := 0;
								arrHPState[1] := 0; arrHPState[2] := 0;
					
	1://Temperature Values from the Heating Pump
	 iStateModbus_CP := iStateModbusRead;
		
		//Reset Write
		fbMBWrite_FC16.bExecute := FALSE;
			
		//Start Read
		fbMBRead_FC4.nQuantity := 16;
			fbMBRead_FC4.nMBAddr := 2002;
				fbMBRead_FC4.bExecute := TRUE;
			
		IF fbMBRead_FC4.bBusy THEN timDelay.IN := TRUE; END_IF
		
		//Wait for Delay, copy Data and then next step
		IF NOT fbMBRead_FC4.bBusy AND NOT fbMBRead_FC4.bError AND timDelay.Q THEN
			//Flow Temp
			fbConvertWordToDword(wInputValue_1:= arrBuffer_FC4[1], wInputValue_2:= arrBuffer_FC4[2], eByteOrderForConvert:= eByteOrder.eLittleEndian, dwOutputValue=> );	
				stFloat.dwRawValue := fbConvertWordToDword.dwOutputValue;
					fbHP.rFlowTemp := stFloat.rValueFloat;
			//Return Temperatur
			fbConvertWordToDword(wInputValue_1:= arrBuffer_FC4[3], wInputValue_2:= arrBuffer_FC4[4], eByteOrderForConvert:= eByteOrder.eLittleEndian, dwOutputValue=> );	
				stFloat.dwRawValue := fbConvertWordToDword.dwOutputValue;
					fbHP.rReturnTemp := stFloat.rValueFloat;
			//Flow Temperature Energy Source
			fbConvertWordToDword(wInputValue_1:= arrBuffer_FC4[5], wInputValue_2:= arrBuffer_FC4[6], eByteOrderForConvert:= eByteOrder.eLittleEndian, dwOutputValue=> );	
				stFloat.dwRawValue := fbConvertWordToDword.dwOutputValue;
					fbHP.rFlowTempEnergySource := stFloat.rValueFloat;
			//Return Temperature Energy Source
			fbConvertWordToDword(wInputValue_1:= arrBuffer_FC4[7], wInputValue_2:= arrBuffer_FC4[8], eByteOrderForConvert:= eByteOrder.eLittleEndian, dwOutputValue=> );	
				stFloat.dwRawValue := fbConvertWordToDword.dwOutputValue;
					fbHP.rReturnTempEnergySource := stFloat.rValueFloat;
			//Boiler Top Temperature for Service Water
			fbConvertWordToDword(wInputValue_1:= arrBuffer_FC4[9], wInputValue_2:= arrBuffer_FC4[10], eByteOrderForConvert:= eByteOrder.eLittleEndian, dwOutputValue=> );	
				stFloat.dwRawValue := fbConvertWordToDword.dwOutputValue;
					fbHP.rBoilerTempServiceWater := stFloat.rValueFloat;
						fbTempS.rRawTempIn := fbHP.rBoilerTempServiceWater;	
			//Boiler Top and Below Temperature for the Heating Boiler
			fbConvertWordToDword(wInputValue_1:= arrBuffer_FC4[13], wInputValue_2:= arrBuffer_FC4[14], eByteOrderForConvert:= eByteOrder.eLittleEndian, dwOutputValue=> );	
				stFloat.dwRawValue := fbConvertWordToDword.dwOutputValue;
					rTB4 := stFloat.rValueFloat;
			fbConvertWordToDword(wInputValue_1:= arrBuffer_FC4[15], wInputValue_2:= arrBuffer_FC4[16], eByteOrderForConvert:= eByteOrder.eLittleEndian, dwOutputValue=> );	
				stFloat.dwRawValue := fbConvertWordToDword.dwOutputValue;
					rTB41 := stFloat.rValueFloat;
 						fbHP.rBoilerTempHeatingSys := (rTB4 + rTB41) / 2;	
			//Go to Next Step
			fbMBRead_FC4.bExecute := FALSE;
				timDelay.IN := FALSE;		
					iStateModbusRead := 2;
		END_IF	

		//Error or Timeout
		IF FPError_FC_4.Q OR timTimeout.Q THEN
			iStateModbusError := 300;
		END_IF
		
	2://Group Error and Error from the Top Temperatursensor in the Service Water Boiler
		iStateModbus_CP := iStateModbusRead;
			
		//Start Read
		fbMBRead_FC4.nQuantity := 13;
			fbMBRead_FC4.nMBAddr := 2210;
				fbMBRead_FC4.bExecute := TRUE;
			
		IF fbMBRead_FC4.bBusy THEN timDelay.IN := TRUE; END_IF
		
		//Wait for Delay, copy Data and then next step
		IF NOT fbMBRead_FC4.bBusy AND NOT fbMBRead_FC4.bError AND timDelay.Q THEN
			//Group Error
			IF arrBuffer_FC4[1] <> 0 THEN bGroupErrorHP := TRUE; ELSE bGroupErrorHP := FALSE; END_IF
			//Alarm index to check if the Temperatursensor in the service water Boiler is ok
			fbConvertWordToDword(wInputValue_1:= arrBuffer_FC4[2], wInputValue_2:= arrBuffer_FC4[3], eByteOrderForConvert:= eByteOrder.eLittleEndian, dwOutputValue=> );	
				arrAlarmList[1] := DWORD_TO_DINT(fbConvertWordToDword.dwOutputValue);
					fbConvertWordToDword(wInputValue_1:= arrBuffer_FC4[4], wInputValue_2:= arrBuffer_FC4[5], eByteOrderForConvert:= eByteOrder.eLittleEndian, dwOutputValue=> );	
						arrAlarmList[2] := DWORD_TO_DINT(fbConvertWordToDword.dwOutputValue);
							fbConvertWordToDword(wInputValue_1:= arrBuffer_FC4[6], wInputValue_2:= arrBuffer_FC4[7], eByteOrderForConvert:= eByteOrder.eLittleEndian, dwOutputValue=> );	
								arrAlarmList[3] := DWORD_TO_DINT(fbConvertWordToDword.dwOutputValue);
			fbConvertWordToDword(wInputValue_1:= arrBuffer_FC4[8], wInputValue_2:= arrBuffer_FC4[9], eByteOrderForConvert:= eByteOrder.eLittleEndian, dwOutputValue=> );	
				arrAlarmList[4] := DWORD_TO_DINT(fbConvertWordToDword.dwOutputValue);						
					fbConvertWordToDword(wInputValue_1:= arrBuffer_FC4[10], wInputValue_2:= arrBuffer_FC4[11], eByteOrderForConvert:= eByteOrder.eLittleEndian, dwOutputValue=> );	
						arrAlarmList[5] := DWORD_TO_DINT(fbConvertWordToDword.dwOutputValue);				
							fbConvertWordToDword(wInputValue_1:= arrBuffer_FC4[12], wInputValue_2:= arrBuffer_FC4[13], eByteOrderForConvert:= eByteOrder.eLittleEndian, dwOutputValue=> );	
								arrAlarmList[6] := DWORD_TO_DINT(fbConvertWordToDword.dwOutputValue);
			IF fbHP.rBoilerTempServiceWater < -90 OR arrAlarmList[1] = 127 OR arrAlarmList[2] = 127 OR arrAlarmList[3] = 127 OR
				arrAlarmList[4] = 127 OR arrAlarmList[5] = 127 OR arrAlarmList[6] = 127 THEN
					bErrorTempSensorBoilerServiceWaterTop := TRUE;
			ELSE
					bErrorTempSensorBoilerServiceWaterTop := FALSE;	
			END_IF
			//Go to Next Step
			fbMBRead_FC4.bExecute := FALSE;
				timDelay.IN := FALSE;		
					iStateModbusRead := 3;
		END_IF	

		//Error or Timeout
		IF FPError_FC_4.Q OR timTimeout.Q THEN
			iStateModbusError := 300;
		END_IF

	3://Heatin Pump "Is running" State
		iStateModbus_CP := iStateModbusRead;

		//Start Read
		fbMBRead_FC4.nQuantity := 4;
			fbMBRead_FC4.nMBAddr := 2030;
				fbMBRead_FC4.bExecute := TRUE;
			
		IF fbMBRead_FC4.bBusy THEN timDelay.IN := TRUE; END_IF
		
		//Wait for Delay, copy Data and then next step
		IF NOT fbMBRead_FC4.bBusy AND NOT fbMBRead_FC4.bError AND timDelay.Q THEN
			//Feedback running
			fbConvertWordToDword(wInputValue_1:= arrBuffer_FC4[1], wInputValue_2:= arrBuffer_FC4[2], eByteOrderForConvert:= eByteOrder.eLittleEndian, dwOutputValue=> );	
				stFloat.dwRawValue := fbConvertWordToDword.dwOutputValue;
					arrHPState[1] := stFloat.rValueFloat;
						fbConvertWordToDword(wInputValue_1:= arrBuffer_FC4[3], wInputValue_2:= arrBuffer_FC4[4], eByteOrderForConvert:= eByteOrder.eLittleEndian, dwOutputValue=> );	
							stFloat.dwRawValue := fbConvertWordToDword.dwOutputValue;
								arrHPState[2] := stFloat.rValueFloat;
			IF arrHPState[1] <> 0 AND arrHPState[2] <> 0 THEN bHPIsRunning := TRUE; ELSE bHPIsRunning := FALSE; END_IF
			//Go to Next Step
			fbMBRead_FC4.bExecute := FALSE;
				timDelay.IN := FALSE;		
					iStateModbusRead := 4;
		END_IF	

		//Error or Timeout
		IF FPError_FC_4.Q OR timTimeout.Q THEN
			iStateModbusError := 300;
		END_IF

	4://Wait 1 Step to reset the delay counter befor start to write
		iStateModbus_CP := iStateModbusRead;
		
		iStateModbusWrite := 1;
			iStateModbusRead := - 1;
				
		//Timeout
		IF timTimeout.Q THEN
			iStateModbusError := 300;
		END_IF	
		
END_CASE		

(*------------------------------------------------------------------Error and Reset----------------------------------------------------------------------------*)	

IF timDissableFunctions.Q THEN fbHP.bWarning := TRUE; fbHP.iWarningCode := 0; ELSE fbHP.bWarning := FALSE; END_IF 	
	IF Lynus_Standards.GVL_Energy.stNumberOfDevices.diNumberOfHP > Constants_Energy.diMaxNumberOfHeatingPumps OR bGroupErrorHP OR fbGetSystemTime.ERR OR bMBTCPError THEN fbHP.bError := TRUE; ELSE fbHP.bError := FALSE; END_IF 

IF Lynus_Standards.GVL_Energy.stNumberOfDevices.diNumberOfHP > Constants_Energy.diMaxNumberOfHeatingPumps THEN fbHP.iErrorCode := 1;
ELSIF fbGetSystemTime.ERR THEN fbHP.iErrorCode := 2; 
ELSIF bGroupErrorHP THEN fbHP.iErrorCode := 0;
ELSIF bMBTCPError THEN fbHP.iErrorCode := 3;
END_IF

FNReset(CLK:= fbHP.stDataHPOut.bSReset, Q=> );
		
//Functionblock HP
fbHP(
	bEnable:= bEnable AND NOT timDissableFunctions.Q,  
	bError:= , 
	bWarning:= , 
	bIsStepSwitched:= FALSE, 
	bEPOIsActive:= , 
	bExternalLock:= fbDIExternalLock.bSignal, 
	bReset:= FNReset.Q, 
	bExternalOnCommand:= Lynus_Standards.GVL_Energy.stDataHeatingPumps[diNrOfEMS_IN,diNrOfHP_OUT].bExternalOnCommand, 
	bWriteWithDelay:= TRUE,
	bHPIsRunning:= bHPIsRunning,
	iErrorCode:= , 
	iWarningCode:= , 
	dwBatterySOC:= , 
	diNumberOfHP:= diNrOfHP_OUT, 
	rBoilerTempHeatingSys:= , 
	rBoilerTempServiceWater:= , 
	rFlowTemp:= , 
	rReturnTemp:= , 
	rFlowTempEnergySource:= , 
	rReturnTempEnergySource:= , 
	lrSizeGridConnection:= lrSizeGridConnection, 
	lrGridPower:= lrGridPower, 
	lrTotalCounterEnergy_Consumption:= , 
	lrTotalCounterEnergy_Production:= , 
	lrCounterEnergyT1_Consumption:= , 
	lrCounterEnergyT2_Consumption:= , 
	lrCounterEnergyT1_Production:= , 
	lrCounterEnergyT2_Production:= , 
	lrCounterThermalEnergy_Heating:= 0, 
	lrCounterThermalEnergy_Water:= 0, 
	lrElPowerHP:= , 
	arrTargetPower:= , 
	tOnDelayExternalOn:= T#2M, 
	tOffDelayExternalOn:= T#2H, 
	tMinOnTime:= T#1H,
	tTimDelayOutput:= T#5S, 
	stSystemTime:= , 
	stSetupHP:= stSetupHP, 
	stDataHPOut=> , 
	stDataHPOutDelay=> stDataHP, 
	arrPercentValuesSteps=> );

(*-------------------------------------------------------------------------Prepear the Output power----------------------------------------------------------------------*)	

rNewPowerToHP := (stSetupHP.rMaxPower1 * fbHP.stDataHPOut.rTargetPower) / 100; 
	rNewPowerToHP := rNewPowerToHP * 1000;
		rNewPowerToHP := LIMIT(0,rNewPowerToHP,100000);	

(*------------------------------------------------------------------Error and Reset Temperature----------------------------------------------------------------------------*)	

IF timDissableFunctions.Q THEN fbTempS.bWarning := TRUE; fbTempS.iWarningCode := 0; ELSE fbTempS.bWarning := FALSE; END_IF   
	IF Lynus_Standards.GVL_Sensors.diNumberOfTemperatureSensors > Constants_Sensors.diMaxNumberOfTemperatureSensors THEN fbTempS.bErrorGeneral := TRUE; fbTempS.iErrorCode := 0; ELSE fbTempS.bErrorGeneral := FALSE; END_IF
		IF bErrorTempSensorBoilerServiceWaterTop OR bMBTCPError THEN fbTempS.usiState.6 := TRUE; ELSE fbTempS.usiState := 0; END_IF
	
//Function Block Temp Sensor Top from the Service Water	
fbTempS(
	bEnable:= bEnable AND NOT timDissableFunctions.Q, 
	bUseFilter:= TRUE, 
	bErrorConfig:= FALSE, 
	bErrorGeneral:= , 
	bWriteWithDelay:= TRUE, 
	usiState:= , 
	iDelayFilter:= 50, 
	iMaxValuesFilter:= 20, 
	iErrorCode:= , 
	iWarningCode:= , 
	rTemperatureOffset:= 0, 
	rRawTempIn:= , 
	tTimDelayOutput:= T#5S, 
	stDataTempOut=> , 
	stDataTempOutDelay=> stDataTempS);

(*------------------------------------------------------------------------------------------State Machine Write---------------------------------------------------------------------------------------------*)	

CASE iStateModbusWrite OF
	
	1://Start with first Register
		iStateModbus_CP := iStateModbusWrite;
		
		fbMBWrite_FC16.nQuantity := 1;
			fbMBWrite_FC16.nMBAddr := 990;
				fbMBWrite_FC16.bExecute := TRUE;
		//Send Value for the Communication handler
		arrBuffer_FC16[1] := 600;
		
		IF fbMBWrite_FC16.bBusy THEN timDelay.IN := TRUE; END_IF

		//Wait for Delay and then next step
		IF NOT fbMBWrite_FC16.bBusy AND NOT fbMBWrite_FC16.bError AND timDelay.Q THEN
			fbMBWrite_FC16.bExecute := FALSE;
				timDelay.IN := FALSE;
					bMBTCPError := FALSE; 
			//Go to Next Step
			iStateModbusWrite := 2;
		END_IF
				
		//Error or Timout
		IF FPError_FC_16.Q OR timTimeout.Q THEN
			iStateModbusError := 300;
		END_IF
		
	2://Next write Register
		iStateModbus_CP := iStateModbusWrite;
		
		fbMBWrite_FC16.nQuantity := 8;
			fbMBWrite_FC16.nMBAddr := 1200;
				fbMBWrite_FC16.bExecute := TRUE;
		//Enable PV Management
		arrBuffer_FC16[1] := 1; arrBuffer_FC16[2] := 0;
		//Enable Surplus Mode
		stFloat.rValueFloat := 1;
			fbConvertDwordToWord(dwInputValue:= stFloat.dwRawValue, eByteOrderForConvert:= eByteOrder.eLittleEndian, wOutputValue_1 => arrBuffer_FC16[3], wOutputValue_2 => arrBuffer_FC16[4]);	
		//Surplus in Watt
		stFloat.rValueFloat := rNewPowerToHP;
			fbConvertDwordToWord(dwInputValue:= stFloat.dwRawValue, eByteOrderForConvert:= eByteOrder.eLittleEndian, wOutputValue_1 => arrBuffer_FC16[5], wOutputValue_2 => arrBuffer_FC16[6]);
		//New Setpoint for Service Water Boiler when PV Management is active
		stFloat.rValueFloat := 62;
			fbConvertDwordToWord(dwInputValue:= stFloat.dwRawValue, eByteOrderForConvert:= eByteOrder.eLittleEndian, wOutputValue_1 => arrBuffer_FC16[5], wOutputValue_2 => arrBuffer_FC16[6]);
		
		IF fbMBWrite_FC16.bBusy THEN timDelay.IN := TRUE; END_IF

		//Wait for Delay and then next step
		IF NOT fbMBWrite_FC16.bBusy AND NOT fbMBWrite_FC16.bError AND timDelay.Q THEN
			fbMBWrite_FC16.bExecute := FALSE;
				timDelay.IN := FALSE;
					bMBTCPError := FALSE; 
						//Restart from new with the Read out part
						iStateModbusRead := 1;
							iStateModbusWrite := 0;
		END_IF
				
		//Error or Timout
		IF FPError_FC_16.Q OR timTimeout.Q THEN
			iStateModbusError := 300;
		END_IF	

END_CASE

(*------------------------------------------------------------------------------------------State Machine Write---------------------------------------------------------------------------------------------*)	

CASE iStateModbusError OF
	
	300://Error
		iStateModbus_CP := iStateModbusError;
			timDelay.IN := FALSE;
				fbMBRead_FC4.bExecute := FALSE;	
					fbMBWrite_FC16.bExecute := FALSE;
						bMBTCPError := TRUE;	
							//Restart from new with the Read out part after an Error
							iStateModbusRead := 1;	
								iStateModbusError := 0;
									iStateModbusWrite := 0;
END_CASE

(*------------------------------------------------------------------------------------------Modbus TCP Functions---------------------------------------------------------------------------------------------*)

fbMBRead_FC4(sIPAddr:= sIPAdress, nUnitID := byUnitID, nTCPPort:= 502, cbLength:= SIZEOF(arrBuffer_FC4), pDestAddr:= ADR(arrBuffer_FC4), tTimeout:= T#10S );
	FPError_FC_4(CLK:= fbMBRead_FC4.bError, Q=> );	
	
fbMBWrite_FC16(sIPAddr:= sIPAdress, nTCPPort:= 502, cbLength:= SIZEOF(arrBuffer_FC16), pSrcAddr:= ADR(arrBuffer_FC16), nUnitID := byUnitID, tTimeout:= T#10S );
	FPError_FC_16(CLK:= fbMBWrite_FC16.bError, Q=> );

(*-----------------------------------------------------------Handle data to Global structure for the heating pump and Temperature Sensor-----------------------------------------------------------------*)

//Delte al old Data on GVL after a online change or change on the variable diNrOfEMS_IDOD
IF diNrOfEMS_IN <> diNrOfEMS_IN_CP AND iStateGVLData = 0 THEN iStateGVLData := 10; END_IF 

CASE iStateGVLData OF
	
	0://Init Step
		byWaitInStep := 0;
			arrCounterForGVL[1] := 1; arrCounterForGVL[2] := 1;
	
	1://Wait for 4 Steps before clean al Data on GVL
		byWaitInStep := byWaitInStep + 1;
			IF byWaitInStep >= 4 AND (fbNumberDevice.bNumberIsCalculatet OR fbNumberDevice_Temp.bNumberIsCalculatet) THEN iStateGVLData := 2; END_IF
				//To much Devices, back to the Init step
				IF byWaitInStep >= 4 AND NOT fbNumberDevice.bNumberIsCalculatet AND NOT fbNumberDevice_Temp.bNumberIsCalculatet THEN iStateGVLData := 0; END_IF	
			
	2://Clear all Data in GVL
		FOR diLPForGVL := 1 TO Constants_Energy.diMaxNumberOfEMS BY 1 DO
			Lynus_Standards.GVL_Energy.stDataHeatingPumps[diLPForGVL,arrCounterForGVL[1]].bEnabled := FALSE;
				Lynus_Standards.GVL_Energy.stDataHeatingPumps[diLPForGVL,arrCounterForGVL[1]].arrMaxPower[1] := 0;
					Lynus_Standards.GVL_Energy.stDataHeatingPumps[diLPForGVL,arrCounterForGVL[1]].arrMaxPower[2] := 0;
						Lynus_Standards.GVL_Energy.stDataHeatingPumps[diLPForGVL,arrCounterForGVL[1]].bIsControllable := FALSE;
							Lynus_Standards.GVL_Energy.stDataHeatingPumps[diLPForGVL,arrCounterForGVL[1]].bIsStepSwitched := FALSE;
								Lynus_Standards.GVL_Energy.stDataHeatingPumps[diLPForGVL,arrCounterForGVL[1]].byErrorWarning := 0;
									Lynus_Standards.GVL_Energy.stDataHeatingPumps[diLPForGVL,arrCounterForGVL[1]].byNumberOfSteps := 0;
										Lynus_Standards.GVL_Energy.stDataHeatingPumps[diLPForGVL,arrCounterForGVL[1]].byPriority := 0;
											Lynus_Standards.GVL_Energy.stDataHeatingPumps[diLPForGVL,arrCounterForGVL[1]].lrElPower := 0;
												Lynus_Standards.GVL_Energy.stDataHeatingPumps[diLPForGVL,arrCounterForGVL[1]].lrElPowerConsumption := 0;
													Lynus_Standards.GVL_Energy.stDataHeatingPumps[diLPForGVL,arrCounterForGVL[1]].lrElPowerProduction := 0;
														Lynus_Standards.GVL_Energy.stDataHeatingPumps[diLPForGVL,arrCounterForGVL[1]].rBoilerTempHeatingSys := 0;
															Lynus_Standards.GVL_Energy.stDataHeatingPumps[diLPForGVL,arrCounterForGVL[1]].rBoilerTempServiceWater := 0;
																Lynus_Standards.GVL_Energy.stDataHeatingPumps[diLPForGVL,arrCounterForGVL[1]].rFlowTemp := 0;
																	Lynus_Standards.GVL_Energy.stDataHeatingPumps[diLPForGVL,arrCounterForGVL[1]].rFlowTempEnergySource := 0;
																		Lynus_Standards.GVL_Energy.stDataHeatingPumps[diLPForGVL,arrCounterForGVL[1]].rReturnTemp := 0;
																			Lynus_Standards.GVL_Energy.stDataHeatingPumps[diLPForGVL,arrCounterForGVL[1]].rReturnTempEnergySource := 0;
																				//Set also the target value from ems back here to 0 and not in EMS function because EMS is in Standy when we have a online change (Problem when we delete a ems function and make a online change)
																				Lynus_Standards.GVL_Energy.stDataHeatingPumps[diLPForGVL,arrCounterForGVL[1]].arrTargetPowerEMS[1] := 0;
																					Lynus_Standards.GVL_Energy.stDataHeatingPumps[diLPForGVL,arrCounterForGVL[1]].arrTargetPowerEMS[2] := 0;
																						Lynus_Standards.GVL_Energy.stDataHeatingPumps[diLPForGVL,arrCounterForGVL[1]].bExternalOnCommand := FALSE;	
		END_FOR
			Lynus_Standards.GVL_Sensors.stDataTemperatureSensors[arrCounterForGVL[2]].bEnabled := FALSE;
				Lynus_Standards.GVL_Sensors.stDataTemperatureSensors[arrCounterForGVL[2]].byErrorWarning := 0;
					Lynus_Standards.GVL_Sensors.stDataTemperatureSensors[arrCounterForGVL[2]].rTemperature := 0;

			//Heating Pumpe		
			arrCounterForGVL[1] := arrCounterForGVL[1] + 1;
				arrCounterForGVL[1] := LIMIT(0,arrCounterForGVL[1],Constants_Energy.diMaxNumberOfHeatingPumps);
			//Temperatur Sensor
			arrCounterForGVL[2] := arrCounterForGVL[2] + 1;
				arrCounterForGVL[2] := LIMIT(0,arrCounterForGVL[2],Constants_Sensors.diMaxNumberOfTemperatureSensors);
					//Back to the init step
					IF arrCounterForGVL[1] >= Constants_Energy.diMaxNumberOfHeatingPumps AND arrCounterForGVL[2] >= Constants_Sensors.diMaxNumberOfTemperatureSensors THEN iStateGVLData := 0; END_IF

	10://Clear old Data on GVL 	
		Lynus_Standards.GVL_Energy.stDataHeatingPumps[diNrOfEMS_IN_CP,diNrOfHP_OUT].bEnabled := FALSE;
			Lynus_Standards.GVL_Energy.stDataHeatingPumps[diNrOfEMS_IN_CP,diNrOfHP_OUT].arrMaxPower[1] := 0;
				Lynus_Standards.GVL_Energy.stDataHeatingPumps[diNrOfEMS_IN_CP,diNrOfHP_OUT].arrMaxPower[2] := 0;
					Lynus_Standards.GVL_Energy.stDataHeatingPumps[diNrOfEMS_IN_CP,diNrOfHP_OUT].bIsControllable := FALSE;
						Lynus_Standards.GVL_Energy.stDataHeatingPumps[diNrOfEMS_IN_CP,diNrOfHP_OUT].bIsStepSwitched := FALSE;
							Lynus_Standards.GVL_Energy.stDataHeatingPumps[diNrOfEMS_IN_CP,diNrOfHP_OUT].byErrorWarning := 0;
								Lynus_Standards.GVL_Energy.stDataHeatingPumps[diNrOfEMS_IN_CP,diNrOfHP_OUT].byNumberOfSteps := 0;
									Lynus_Standards.GVL_Energy.stDataHeatingPumps[diNrOfEMS_IN_CP,diNrOfHP_OUT].byPriority := 0;
										Lynus_Standards.GVL_Energy.stDataHeatingPumps[diNrOfEMS_IN_CP,diNrOfHP_OUT].lrElPower := 0;
											Lynus_Standards.GVL_Energy.stDataHeatingPumps[diNrOfEMS_IN_CP,diNrOfHP_OUT].lrElPowerConsumption := 0;
												Lynus_Standards.GVL_Energy.stDataHeatingPumps[diNrOfEMS_IN_CP,diNrOfHP_OUT].lrElPowerProduction := 0;
													Lynus_Standards.GVL_Energy.stDataHeatingPumps[diNrOfEMS_IN_CP,diNrOfHP_OUT].rBoilerTempHeatingSys := 0;
														Lynus_Standards.GVL_Energy.stDataHeatingPumps[diNrOfEMS_IN_CP,diNrOfHP_OUT].rBoilerTempServiceWater := 0;
															Lynus_Standards.GVL_Energy.stDataHeatingPumps[diNrOfEMS_IN_CP,diNrOfHP_OUT].rFlowTemp := 0;
																Lynus_Standards.GVL_Energy.stDataHeatingPumps[diNrOfEMS_IN_CP,diNrOfHP_OUT].rFlowTempEnergySource := 0;
																	Lynus_Standards.GVL_Energy.stDataHeatingPumps[diNrOfEMS_IN_CP,diNrOfHP_OUT].rReturnTemp := 0;
																		Lynus_Standards.GVL_Energy.stDataHeatingPumps[diNrOfEMS_IN_CP,diNrOfHP_OUT].rReturnTempEnergySource := 0;										
		diNrOfEMS_IN_CP := diNrOfEMS_IN;
			//Back to the init step
			iStateGVLData := 0;

END_CASE 	 

IF diNrOfHP_OUT > 0 AND fbNumberDevice.bNumberIsCalculatet AND diNrOfEMS_IN > 0 THEN
	Lynus_Standards.GVL_Energy.stDataHeatingPumps[diNrOfEMS_IN,diNrOfHP_OUT].bEnabled := fbHP.stDataHPOut.bEnabled;
		Lynus_Standards.GVL_Energy.stDataHeatingPumps[diNrOfEMS_IN,diNrOfHP_OUT].arrMaxPower[1] := fbHP.stDataHPOut.arrMaxPower[1];
			Lynus_Standards.GVL_Energy.stDataHeatingPumps[diNrOfEMS_IN,diNrOfHP_OUT].arrMaxPower[2] := fbHP.stDataHPOut.arrMaxPower[2];
				Lynus_Standards.GVL_Energy.stDataHeatingPumps[diNrOfEMS_IN,diNrOfHP_OUT].bIsControllable := TRUE;
					Lynus_Standards.GVL_Energy.stDataHeatingPumps[diNrOfEMS_IN,diNrOfHP_OUT].bIsStepSwitched := fbHP.stDataHPOut.bIsStepSwitched;
						Lynus_Standards.GVL_Energy.stDataHeatingPumps[diNrOfEMS_IN,diNrOfHP_OUT].byErrorWarning := fbHP.stDataHPOut.byErrorWarning;
							Lynus_Standards.GVL_Energy.stDataHeatingPumps[diNrOfEMS_IN,diNrOfHP_OUT].byNumberOfSteps := fbHP.stDataHPOut.byNumberOfSteps;
								Lynus_Standards.GVL_Energy.stDataHeatingPumps[diNrOfEMS_IN,diNrOfHP_OUT].byPriority := fbHP.stDataHPOut.byPriority;
									Lynus_Standards.GVL_Energy.stDataHeatingPumps[diNrOfEMS_IN,diNrOfHP_OUT].lrElPower := fbHP.stDataHPOut.lrElPower;
										Lynus_Standards.GVL_Energy.stDataHeatingPumps[diNrOfEMS_IN,diNrOfHP_OUT].lrElPowerConsumption := fbHP.stDataHPOut.lrElPowerConsumption;
											Lynus_Standards.GVL_Energy.stDataHeatingPumps[diNrOfEMS_IN,diNrOfHP_OUT].lrElPowerProduction := fbHP.stDataHPOut.lrElPowerProduction;
												Lynus_Standards.GVL_Energy.stDataHeatingPumps[diNrOfEMS_IN,diNrOfHP_OUT].rBoilerTempHeatingSys := fbHP.stDataHPOut.rBoilerTempHeatingSys;
													Lynus_Standards.GVL_Energy.stDataHeatingPumps[diNrOfEMS_IN,diNrOfHP_OUT].rBoilerTempServiceWater := fbHP.stDataHPOut.rBoilerTempServiceWater;
														Lynus_Standards.GVL_Energy.stDataHeatingPumps[diNrOfEMS_IN,diNrOfHP_OUT].rFlowTemp := fbHP.stDataHPOut.rFlowTemp;
															Lynus_Standards.GVL_Energy.stDataHeatingPumps[diNrOfEMS_IN,diNrOfHP_OUT].rFlowTempEnergySource := fbHP.stDataHPOut.rFlowTempEnergySource;
																Lynus_Standards.GVL_Energy.stDataHeatingPumps[diNrOfEMS_IN,diNrOfHP_OUT].rReturnTemp := fbHP.stDataHPOut.rReturnTemp;
																	Lynus_Standards.GVL_Energy.stDataHeatingPumps[diNrOfEMS_IN,diNrOfHP_OUT].rReturnTempEnergySource := fbHP.stDataHPOut.rReturnTempEnergySource;	
END_IF

IF diNrOfTempS_OUT_ServiceWaterTop > 0 AND fbNumberDevice_Temp.bNumberIsCalculatet THEN
	Lynus_Standards.GVL_Sensors.stDataTemperatureSensors[diNrOfTempS_OUT_ServiceWaterTop].bEnabled := fbTempS.stDataTempOut.bEnabled;
		Lynus_Standards.GVL_Sensors.stDataTemperatureSensors[diNrOfTempS_OUT_ServiceWaterTop].byErrorWarning := fbTempS.stDataTempOut.byErrorWarning;
			Lynus_Standards.GVL_Sensors.stDataTemperatureSensors[diNrOfTempS_OUT_ServiceWaterTop].rTemperature := fbTempS.stDataTempOut.rTemperature;
END_IF

(*----------------------------------------------------------Save persistent data----------------------------------------------------------------*)

arrPD[1](lrValue:= BOOL_TO_LREAL(bEnable), bEventBasedActive=> );
arrPD[2](lrValue:= BOOL_TO_LREAL(bPowerDataInvers), bEventBasedActive=> );
arrPD[3](lrValue:= DINT_TO_LREAL(diNrOfEMS_IN), bEventBasedActive=> );
arrPD[4](lrValue:= DINT_TO_LREAL(diNrOfEM_IN_HP), bEventBasedActive=> );
arrPD[5](lrValue:= DINT_TO_LREAL(diNrOfEMS_IN_CP), bEventBasedActive=> );
arrPD[6](lrValue:= REAL_TO_LREAL(stSetupHP.rMaxPower1), bEventBasedActive=> );
arrPD[7](lrValue:= REAL_TO_LREAL(stSetupHP.rMaxPower2), bEventBasedActive=> );
arrPD[8](lrValue:= BOOL_TO_LREAL(stSetupHP.bManualyOn), bEventBasedActive=> );
arrPD[9](lrValue:= BOOL_TO_LREAL(stSetupHP.bOnEmergPowerOff), bEventBasedActive=> );
arrPD[10](lrValue:= BOOL_TO_LREAL(stSetupHP.bOnEmergPowerOff), bEventBasedActive=> );
arrPD[11](lrValue:= BOOL_TO_LREAL(stSetupHP.bTimeEnabled), bEventBasedActive=> );
arrPD[12](lrValue:= BYTE_TO_LREAL(stSetupHP.byDisableSOC), bEventBasedActive=> );
arrPD[13](lrValue:= BYTE_TO_LREAL(stSetupHP.byEnableSOC), bEventBasedActive=> );
arrPD[14](lrValue:= BYTE_TO_LREAL(stSetupHP.byHourOff), bEventBasedActive=> );
arrPD[15](lrValue:= BYTE_TO_LREAL(stSetupHP.byHourOn), bEventBasedActive=> );
arrPD[16](lrValue:= BYTE_TO_LREAL(stSetupHP.byManualyTargetPower), bEventBasedActive=> );
arrPD[17](lrValue:= BYTE_TO_LREAL(stSetupHP.byMinutesOff), bEventBasedActive=> );
arrPD[18](lrValue:= BYTE_TO_LREAL(stSetupHP.byMinutesOn), bEventBasedActive=> );
arrPD[19](lrValue:= BYTE_TO_LREAL(stSetupHP.byPriority), bEventBasedActive=> );
arrPD[20](lrValue:= BYTE_TO_LREAL(stSetupHP.byTimeEnabledTargetPower), bEventBasedActive=> );
arrPD[21](lrValue:= BYTE_TO_LREAL(byUnitID), bEventBasedActive=> );
fbPDString(sText:= sIPAdress, bEventBasedActive=> );

END_FUNCTION_BLOCK

// ---- FBs/EconSolutions/FB_EconSens3.TcPOU
FUNCTION_BLOCK FB_EconSens3
VAR_INPUT PERSISTENT
	m_Enable					: BOOL;						//Enable the Fuctionblock and his logic
	str_IPAdress				: STRING(15);				//IP Adress of the meter
END_VAR
VAR_OUTPUT
	real_RealPower_kW				: REAL;					// Real power in kW
	real_RealPowerL1_kW				: REAL;					// Real power in kW
	real_RealPowerL2_kW				: REAL;					// Real power in kW
	real_RealPowerL3_kW				: REAL;					// Real power in kW
	real_ReactivePower_kVAr			: REAL;					// Reactive power in kVAr
	real_ReactivePowerL1_kVAr		: REAL;					// Reactive power in kVAr
	real_ReactivePowerL2_kVAr		: REAL;					// Reactive power in kVAr
	real_ReactivePowerL3_kVAr		: REAL;					// Reactive power in kVAr
	real_ApparentPower_kVA			: REAL;					// Apparent power in kVA
	real_ApparentPowerL1_kVA			: REAL;					// Apparent power in kVA
	real_ApparentPowerL2_kVA			: REAL;					// Apparent power in kVA
	real_ApparentPowerL3_kVA			: REAL;					// Apparent power in kVA
	real_Frequency_Hz				: REAL;					// Frequency in Hz
	real_VoltageL1N_V				: REAL;					//  Voltage L1-N in V 
	real_VoltageL2N_V				: REAL;					//  Voltage L2-N in V 
	real_VoltageL3N_V				: REAL;					//  Voltage L3-N in V 
	real_VoltageL1L2_V				: REAL;					//  Voltage L1-L2 in V 
	real_VoltageL2L3_V				: REAL;					//  Voltage L2-L3 in V 
	real_VoltageL3L1_V				: REAL;					//  Voltage L3-L1 in V 
	real_CurrentL1_A				: REAL;					//  Current L1 in A
	real_CurrentL2_A				: REAL;					//  Current L2 in A
	real_CurrentL3_A				: REAL;					//  Current L3 in A
	real_EnergyTotal_Import_kWh		: REAL;					// Energy total in kWh
	real_EnergyTotal_Export_kWh		: REAL;					// Energy total in kWh
	real_Temperatur_C				: REAL;					//  Temperatur in °C
	
	m_PollSuccessful				: BOOL;					// Poll succesfull		
	udint_Error_ID					: UDINT;				// ERR ID FB_MBReadRegs
END_VAR
VAR
//	{attribute 'hide'}
	w_Adress					: WORD;						//modbus adress
//	{attribute 'hide'}
	usint_Quantity				: USINT;					//Number of Words to get polled, max 100
//	{attribute 'hide'}
	fb_Convert_Data				: FB_Convert_Dword_Real;
//	{attribute 'hide'}
	e_ByteOrderConvert			: eByteOrder;						//Byte Format
//	{attribute 'hide'}
	timer_Delay					: TON;						//Timer for Delay between Requests
//	{attribute 'hide'}
	timer_DelayStart			: TON;						//Timer to start the state machine with Delay after enabling or after the system ist restartet
//	{attribute 'hide'}
	timer_TimeOut				: TON;						//Timer for Timeout MB Read
//	{attribute 'hide'}
	iStateModbusRead			: INT;						//State machine for read out Data over Modbus RTU
//	{attribute 'hide'}
	fbMBRead_FC3				: FB_MBReadRegs  ;		//Modbus Read Function (FC3)
//	{attribute 'hide'}
	ftrig_PEnable				: f_trig;					//Internal positive Edge
//	{attribute 'hide'}
	iStateModbusError			: INT;						//State machine for error out Data over Modbus TCP/IP	
//	{attribute 'hide'}
	FPError_FC_3				: R_TRIG;					//Internal positive Edge
//	{attribute 'hide'}
	arrBuffer_FC3				: ARRAY[0..100] OF WORD;		//Buffer with Data from FC3
//	{attribute 'hide'}
	arrBuffer_Received			: ARRAY[1..2,0..100] OF WORD;		//Total received Data
//	{attribute 'hide'}
	timer_Connection_ok			: TON;
//	{attribute 'hide'}
	int_Data_Received			: INT;
//	{attribute 'hide'}
	m_MBTCPError				: BOOL;
//	{attribute 'hide'}
	int_Data_Received_old		: INT;
//	{attribute 'hide'}
	timer_Connection_ok_TOF	: TOF;
//	{attribute 'hide'}
	m_Poll_ok: BOOL;
//	{attribute 'hide'}
	timer_Wait: Ton;
//	{attribute 'hide'}
	int_TimeoutError: INT;
//	{attribute 'hide'}
	int_FC4Error: INT;
//	{attribute 'hide'}
	i: INT;
//	{attribute 'hide'}
	x: INT;
//	{attribute 'hide'}
	time_wait: TIME:=T#1S;
END_VAR

// v0.1 by Stefan Lackner 20230729
// untested
// reads out EconSolution EconSens3 Multimeter


(*--------------------------------------------------------------------------------------------Limits-------------------------------------------------------------------------------------*)
w_Adress := LIMIT(0,w_Adress,65000);
usint_Quantity := LIMIT(1,usint_Quantity,100);
	
(*--------------------------------------------------------------------------------------------State Machine Read--------------------------------------------------------------------------------------*)

//Timer for Delay
timer_Delay(IN:= , PT:= T#50MS, Q=> , ET=> );

//Timeout Timer is dissabled when the Init Step is aktiv or the function is not enabled
IF iStateModbusRead = 0 OR NOT m_Enable THEN 
	timer_Timeout.IN := FALSE; 
END_IF
timer_Timeout(IN:= , PT:= T#1S, Q=> , ET=> );

//Enable with Delay that not all sockets have to be created at the same time
timer_DelayStart(IN:= m_Enable, PT:= T#1S, Q=> , ET=> );
ftrig_PEnable(CLK:= timer_DelayStart.Q, Q=> );

IF ftrig_PEnable.Q AND iStateModbusRead = 0 THEN 
	iStateModbusRead := 1; 
END_IF		
		
//Not Enabled
IF NOT m_Enable THEN 
	iStateModbusRead := 0; 
	iStateModbusError := 0; 
END_IF		
		
CASE iStateModbusRead OF

	0://Init Step 
		timer_Delay.IN := FALSE;
		fbMBRead_FC3.bExecute := FALSE;
		m_Poll_ok:=FALSE;
		int_Data_Received:=0;
		iStateModbusRead := iStateModbusRead+1;

	1: // clean the array  Poll 1
		FOR i:=0 TO 100 BY 1 DO
			arrBuffer_FC3[i] := 0;
		END_FOR
		w_Adress := 17;
		usint_Quantity := 94; 
		iStateModbusRead := iStateModbusRead+1;
		
	2://read the required registers
		//Start Read Poll 1
		fbMBRead_FC3.nQuantity := usint_Quantity;
		fbMBRead_FC3.nMBAddr := w_Adress;
		fbMBRead_FC3.bExecute := TRUE;
		fbMBRead_FC3.nUnitID := 1;
		timer_Timeout.IN := TRUE;
		IF fbMBRead_FC3.bBusy THEN 
			timer_Delay.IN := TRUE; 
		END_IF
		
		//Wait for Delay, copy Data and then next step
		IF NOT fbMBRead_FC3.bBusy AND NOT fbMBRead_FC3.bError AND timer_Delay.Q THEN
			m_Poll_ok:=TRUE;
			int_Data_Received:=int_Data_Received+1;
			m_MBTCPError := FALSE; 
			
			FOR i:=0 TO 100 BY 1 DO
				arrBuffer_Received[1,i] := arrBuffer_FC3[i];
			END_FOR
			
			//Go to Next Step
			timer_Timeout.IN := FALSE;
			fbMBRead_FC3.bExecute := FALSE;
			timer_Delay.IN := FALSE;		
			iStateModbusRead := 30;
		END_IF	

		//Error or Timeout
		IF FPError_FC_3.Q THEN 
			iStateModbusError := 300;
			int_FC4Error := int_FC4Error+1;
		ELSIF timer_Timeout.Q THEN  
			timer_Timeout.IN := FALSE; 	
			iStateModbusError := 300;
			int_TimeoutError := int_TimeoutError+1;
		END_IF
	
	
	30: // convert data
		e_ByteOrderConvert := 0;			// 		eBigEndian	:= 0,  eLittleEndian	:= 1
		x:=0;
		fb_Convert_Data(	word_In_1:= arrBuffer_Received[1,x], 
							word_In_2:= arrBuffer_Received[1,x+1], 
							e_ByteOrderIn:= e_ByteOrderConvert, 
							real_Output=> real_VoltageL1L2_V);
		x:=x+2;
		fb_Convert_Data(	word_In_1:= arrBuffer_Received[1,x], 
							word_In_2:= arrBuffer_Received[1,x+1], 
							e_ByteOrderIn:= e_ByteOrderConvert, 
							real_Output=> real_VoltageL2L3_V);
		x:=x+2;
		fb_Convert_Data(	word_In_1:= arrBuffer_Received[1,x], 
							word_In_2:= arrBuffer_Received[1,x+1], 
							e_ByteOrderIn:= e_ByteOrderConvert, 
							real_Output=> real_VoltageL3L1_V);		
		x:=x+2;
		fb_Convert_Data(	word_In_1:= arrBuffer_Received[1,x], 
							word_In_2:= arrBuffer_Received[1,x+1], 
							e_ByteOrderIn:= e_ByteOrderConvert, 
							real_Output=> real_VoltageL1N_V);
		x:=x+2;
		fb_Convert_Data(	word_In_1:= arrBuffer_Received[1,x], 
							word_In_2:= arrBuffer_Received[1,x+1], 
							e_ByteOrderIn:= e_ByteOrderConvert, 
							real_Output=> real_VoltageL2N_V);
		x:=x+2;
		fb_Convert_Data(	word_In_1:= arrBuffer_Received[1,x], 
							word_In_2:= arrBuffer_Received[1,x+1], 
							e_ByteOrderIn:= e_ByteOrderConvert, 
							real_Output=> real_VoltageL3N_V);
		x:=x+2;
		fb_Convert_Data(	word_In_1:= arrBuffer_Received[1,x], 
							word_In_2:= arrBuffer_Received[1,x+1], 
							e_ByteOrderIn:= e_ByteOrderConvert, 
							real_Output=> real_CurrentL1_A);
		x:=x+2;
		fb_Convert_Data(	word_In_1:= arrBuffer_Received[1,x], 
							word_In_2:= arrBuffer_Received[1,x+1], 
							e_ByteOrderIn:= e_ByteOrderConvert, 
							real_Output=> real_CurrentL2_A);
		x:=x+2;
		fb_Convert_Data(	word_In_1:= arrBuffer_Received[1,x], 
							word_In_2:= arrBuffer_Received[1,x+1], 
							e_ByteOrderIn:= e_ByteOrderConvert, 
							real_Output=> real_CurrentL3_A);		
		x:=x+2;
		fb_Convert_Data(	word_In_1:= arrBuffer_Received[1,x], 
							word_In_2:= arrBuffer_Received[1,x+1], 
							e_ByteOrderIn:= e_ByteOrderConvert, 
							real_Output=> real_RealPowerL1_kW);
		x:=x+2;		
		fb_Convert_Data(	word_In_1:= arrBuffer_Received[1,x], 
							word_In_2:= arrBuffer_Received[1,x+1], 
							e_ByteOrderIn:= e_ByteOrderConvert, 
							real_Output=> real_RealPowerL2_kW);		
		x:=x+2;		
		fb_Convert_Data(	word_In_1:= arrBuffer_Received[1,x], 
							word_In_2:= arrBuffer_Received[1,x+1], 
							e_ByteOrderIn:= e_ByteOrderConvert, 
							real_Output=> real_RealPowerL3_kW);	
		x:=x+2;		
		fb_Convert_Data(	word_In_1:= arrBuffer_Received[1,x], 
							word_In_2:= arrBuffer_Received[1,x+1], 
							e_ByteOrderIn:= e_ByteOrderConvert, 
							real_Output=> real_ReactivePowerL1_kVAr);	
		x:=x+2;		
		fb_Convert_Data(	word_In_1:= arrBuffer_Received[1,x], 
							word_In_2:= arrBuffer_Received[1,x+1], 
							e_ByteOrderIn:= e_ByteOrderConvert, 
							real_Output=> real_ReactivePowerL2_kVAr);	
		x:=x+2;		
		fb_Convert_Data(	word_In_1:= arrBuffer_Received[1,x], 
							word_In_2:= arrBuffer_Received[1,x+1], 
							e_ByteOrderIn:= e_ByteOrderConvert, 
							real_Output=> real_ReactivePowerL3_kVAr);
		x:=x+2;		
		fb_Convert_Data(	word_In_1:= arrBuffer_Received[1,x], 
							word_In_2:= arrBuffer_Received[1,x+1], 
							e_ByteOrderIn:= e_ByteOrderConvert, 
							real_Output=> real_ApparentPowerL1_kVA);	
		x:=x+2;		
		fb_Convert_Data(	word_In_1:= arrBuffer_Received[1,x], 
							word_In_2:= arrBuffer_Received[1,x+1], 
							e_ByteOrderIn:= e_ByteOrderConvert, 
							real_Output=> real_ApparentPowerL2_kVA);	
		x:=x+2;		
		fb_Convert_Data(	word_In_1:= arrBuffer_Received[1,x], 
							word_In_2:= arrBuffer_Received[1,x+1], 
							e_ByteOrderIn:= e_ByteOrderConvert, 
							real_Output=> real_ApparentPowerL3_kVA);		
		real_RealPower_kW := real_RealPowerL1_kW +real_RealPowerL2_kW + real_RealPowerL3_kW;
		real_ReactivePower_kVAr := real_ReactivePowerL1_kVAr + real_ReactivePowerL2_kVAr + real_ReactivePowerL3_kVAr;
 		real_ApparentPower_kVA := real_ApparentPowerL1_kVA + real_ApparentPowerL2_kVA + real_ApparentPowerL3_kVA;

		x:=56;		
		fb_Convert_Data(	word_In_1:= arrBuffer_Received[1,x], 
							word_In_2:= arrBuffer_Received[1,x+1], 
							e_ByteOrderIn:= e_ByteOrderConvert, 
							real_Output=> real_Temperatur_C);		
		x:=58;		
		fb_Convert_Data(	word_In_1:= arrBuffer_Received[1,x], 
							word_In_2:= arrBuffer_Received[1,x+1], 
							e_ByteOrderIn:= e_ByteOrderConvert, 
							real_Output=> real_Frequency_Hz);									
	
			
		x:=60;	
		fb_Convert_Data(	word_In_1:= arrBuffer_Received[1,x], 
							word_In_2:= arrBuffer_Received[1,x+1], 
							e_ByteOrderIn:= e_ByteOrderConvert, 
							real_Output=> real_EnergyTotal_Import_kWh);		
		x:=68;	
		fb_Convert_Data(	word_In_1:= arrBuffer_Received[1,x], 
							word_In_2:= arrBuffer_Received[1,x+1], 
							e_ByteOrderIn:= e_ByteOrderConvert, 
							real_Output=> real_EnergyTotal_Export_kWh);		
		
		// go to next state
		iStateModbusRead := iStateModbusRead+1;		
		
	31://Wait and go to start
		timer_Wait.IN := TRUE;
		
		IF timer_Wait.Q = TRUE THEN
			iStateModbusRead := 1;
			timer_Wait.IN :=FALSE;
		END_IF	

END_CASE

(* wait timer*)

timer_Wait(PT:=time_wait);


(*------------------------------------------------------------------Error and Warning----------------------------------------------------------------------------*)	
 
timer_Connection_ok			(In:=int_Data_Received<>int_Data_Received_old,PT:=T#10S);
timer_Connection_ok_TOF		(In:=NOT(int_Data_Received<>int_Data_Received_old) AND int_Data_Received>3 ,PT:=T#20S);
int_Data_Received_old:=int_Data_Received;
m_PollSuccessful:=NOT timer_Connection_ok.Q AND timer_Connection_ok_TOF.Q ;

(*------------------------------------------------------------------------------------------Modbus TCP Functions---------------------------------------------------------------------------------------------*)

fbMBRead_FC3(	sIPAddr:= str_IPAdress, 
				nTCPPort:= 502,
				cbLength:= SIZEOF(arrBuffer_FC3), 
				pDestAddr:= ADR(arrBuffer_FC3), 
				tTimeout:= T#10S,
				nErrId => udint_Error_ID);

FPError_FC_3(CLK:= fbMBRead_FC3.bError, Q=> );		

(*------------------------------------------------------------------------------------------State Machine Error---------------------------------------------------------------------------------------------*)	

CASE iStateModbusError OF
	
	300://Error
		timer_Wait.IN :=TRUE;
		timer_Delay.IN := FALSE;
		fbMBRead_FC3.bExecute := FALSE;
		m_MBTCPError := TRUE; 		
		m_Poll_ok:=FALSE;
		int_Data_Received:=0;
		
				//Restart from new with the Read out part after an Error
		IF timer_Wait.Q = TRUE THEN
			iStateModbusRead := 0;	
			iStateModbusError := 0;
			timer_Wait.IN :=FALSE;
			timer_Timeout.IN := FALSE;
		END_IF		
							
END_CASE

END_FUNCTION_BLOCK

// ---- FBs/Firmer/FB_Firmer_PV_Inverter_Sunspec.TcPOU
FUNCTION_BLOCK FB_Firmer_PV_Inverter_Sunspec
VAR_INPUT PERSISTENT
	///{#lynus.ag#()} //Enable the Fuctionblock and his logic
	bEnable: BOOL;
	///Unit ID for the Inverter
	byUnitID_Inverter: BYTE;
	///IP Adress from the Inverter
	sIPAdress: STRING(15);
END_VAR
VAR_OUTPUT
	///Structure with specific Firmer Inverter Data
	stFirmerInverterData: ST_FirmerPvInverter_Data;
	///Output structure with Data from Electric Meter PV (Power Data)
	stDataEMPower_PV: ST_ElectricMeter_Output_Power;
	///Output structure with Data from Electric Meter PV (Counter Data)
	stDataEMCounter_PV: ST_ElectricMeter_Output_Counter;
	///Active Number from the Electric Meter for using on other functions
	diNrOfEM_OUT_PV: DINT;
END_VAR
VAR
	///Electric Meter Function 
	{attribute 'hide' := ''}
	fbElMeter: FB_ElectricMeter;
	///Function block to calcualte the number of the Device
	{attribute 'hide' := ''}
	fbNumberDevice: FB_NumberOfDevice;
	///Modbus Read Function (FC3)
	{attribute 'hide' := ''}
	fbMBRead_FC3: FB_MBReadRegs;
	///Timer for Delay between Requests
	{attribute 'hide' := ''}
	timDelay: TON;
	///Timer for Timeout
	{attribute 'hide' := ''}
	timTimeout: TON;
	///Timer to dissable the Function after Lynus_Standards.Constants_General.tTimeDissableLynusFunctions Days without connection to the Lynus Cloud
	{attribute 'hide' := ''}
	timDissableFunctions: TON;
	///Timer to try reset the connection Flag on the GVL. (When somebody delete the Connection Function and make only a onlinechange)
	{attribute 'hide' := ''}
	timResetConnectionOnGVL: TON;
	///Timer to Close the Socket after to much Errors
	{attribute 'hide' := ''}
	timCloseSocket: TON;
	///Internal positive Edge
	{attribute 'hide' := ''}
	FPEnable: R_TRIG;
	///Internal positive Edge
	{attribute 'hide' := ''}
	FPError_FC_3: R_TRIG;
	///Convert 2 WORD in a DWORD
	{attribute 'hide' := ''}
	fbConvertWord: FB_CV_WORD_TO_DWORD;
	///Function to save persistent string data
	{attribute 'hide' := ''}
	fbPDString: FB_PersistentData_String;
	///Function to save persistent data
	{attribute 'hide' := ''}
	arrPD: ARRAY[1..2] OF FB_PersistentData_Number;
	///Buffer with Data from FC3
	{attribute 'hide' := ''}
	arrBuffer_FC3: ARRAY[1..120] OF WORD;
	///Error or Fault from Inverter
	{attribute 'hide' := ''}
	bErrorInverter: BOOL;
	///Error Counter when we have TCP Error or Timeout Error
	{attribute 'hide' := ''}
	byErrorCounterTCP: BYTE;
	///Wait in Step before start to clean data on PLC
	{attribute 'hide' := ''}
	byWaitInStep: BYTE;
	///Variable for Loop to fill default values in the Firmer output structure
	{attribute 'hide' := ''}
	byLPFillDefaultData: BYTE;
	///State machine to handle the data on the GVL
	{attribute 'hide' := ''}
	iStateGVLData: INT;
	///State machine for read out Data over Modbus RTU
	{attribute 'hide' := ''}
	iStateModbusRead: INT;
	///State machine for error out Data over Modbus RTU	
	{attribute 'hide' := ''}
	iStateModbusError: INT;
	///Variable to compare the state machine variable to set or reset the timeout timer
	{attribute 'hide' := ''}
	iStateModbus_CP: INT;
	///Scale Factor for MPPT Power
	{attribute 'hide' := ''}
	iSFPowerMPPT: INT;
	///Number of MPPT
	{attribute 'hide' := ''}
	wNumberOfMPPT: WORD;
	///Variable for Loop to fill the power for each MPPT in the output structure
	{attribute 'hide' := ''}
	wLPPowerMPPT: WORD;
	///Next Modbus Start Adress why in Pic 160 the Number of Registers is variabel and so the next Modbus Registers in the next Pics can be different
	{attribute 'hide' := ''}
	wNextModbusStartAdress: WORD;
	///Number of Inputs from Pic 401 to calculate the Next Modbus Start Adress
	{attribute 'hide' := ''}
	wNumberOfInputs: WORD;
	///ID of the PIC
	{attribute 'hide' := ''}
	wPicID: WORD;
	///Counter to clean old data on GVL
	{attribute 'hide' := ''}
	diCounterForGVL: DINT;
	///Rest of the calculation for new Star Adress. In Sunspec each new PIC start with a even adress
	{attribute 'hide' := ''}
	lrRestNextAdress: LREAL;
END_VAR

//Creator : Kai Ebensperger
//Company : Lynus AG
//Date : 19.07.2022
//Version : 1.0.0.0

//With this function its possible to read out values from the Firmer PV Inverter over Modbus TCP
//The Protocoll is the Sunspec Protocol
//Versions that are supported : 1.0.11
//This Function use the INT + Scalfactor Format

//NOTE for diNr.....Designation => 
//_IN = Here Data come in from other Functions or go out to other functions about the GVL
//_OUT = Here Data go out to other functions about the GVL

(*-------------------------------------------------------------Calcualte the number of ECS---------------------------------------------------------------*)

fbNumberDevice(
	diActualNumberOfDevices:= Lynus_Standards.GVL_Energy.stNumberOfDevices.diNumberOfElectricMeters, 
	diMaxNumberOfDevices:= Constants_Energy.diMaxNumberOfElectricMeters, 
	udiCounterOnlineChange:= TwinCAT_SystemInfoVarList._AppInfo.OnlineChangeCnt, 
	bNumberIsCalculatet=> , 
	bFPNumberIsCalculatet=> , 
	bOnlineChange=> , 
	diNumberForThisDevice=> diNrOfEM_OUT_PV, 
	diNumberOfTotalDevices=> );

//Write new Numer on GVL
IF fbNumberDevice.bFPNumberIsCalculatet THEN
	Lynus_Standards.GVL_Energy.stNumberOfDevices.diNumberOfElectricMeters := fbNumberDevice.diNumberOfTotalDevices;	
END_IF 

//Delete old Number on GVL
IF fbNumberDevice.bOnlineChange THEN 
	Lynus_Standards.GVL_Energy.stNumberOfDevices.diNumberOfElectricMeters := diNrOfEM_OUT_PV;	
		iStateGVLData := 1;
END_IF

(*-------------------------------------------------------------Service from Backend is ready and check the connection to backen for dissabel/enable Function---------------------------------------------------------------*)

//Try to reset the variable for connection on the GVL. When all is normal then the Lynus Mqtt connection function set this variable to true in the next cycle
//When we have no connection to the backend then after Lynus_Standards.Constants_General.tTimeDissableLynusFunctions days the Function is dissabled with all of his functionalities
timResetConnectionOnGVL(IN:= NOT timResetConnectionOnGVL.Q, PT:= T#1H, Q=> , ET=> );
	IF timResetConnectionOnGVL.Q THEN Lynus_Standards.GVL_Communicator.bStateConnectionToEnableFunctions := FALSE; END_IF
		IF NOT Lynus_Standards.GVL_Communicator.bStateConnectionToEnableFunctions THEN timDissableFunctions.IN := TRUE; ELSE timDissableFunctions.IN := FALSE; END_IF  
			timDissableFunctions(IN:= , PT:= Lynus_Standards.Constants_General.tTimeDissableLynusFunctions, Q=> , ET=> );
			
(*--------------------------------------------------------------------------------------------State Machine Read--------------------------------------------------------------------------------------*)

//Timer for Delay
timDelay(IN:= , PT:= T#250MS, Q=> , ET=> );

//Timer for Timeout in Statemachine
IF iStateModbusRead > 0 AND iStateModbusRead <= 5 AND iStateModbusRead = iStateModbus_CP THEN
		timTimeout.IN := TRUE;
ELSE	
		timTimeout.IN := FALSE;
END_IF
	//Timeout Timer is dissabled when the slave wait that his adress is in porgress on the RTU Master, or is dissabled or the Terminal is not configured
	IF iStateModbusRead = 0 OR NOT bEnable THEN timTimeout.IN := FALSE; END_IF
		timTimeout(IN:= , PT:= T#15S, Q=> , ET=> );

//Enable the State Machine
FPEnable(CLK:= bEnable, Q=> );
	IF FPEnable.Q AND iStateModbusRead = 0 THEN iStateModbusRead := 1; END_IF		
		
//Not Enabled
IF NOT bEnable THEN iStateModbusRead := 0; iStateModbusError := 0; END_IF		
		
CASE iStateModbusRead OF

	0://Init Step (Wait that the Slave is enabled and the Terminal is configured)
		iStateModbus_CP := 0;
			timDelay.IN := FALSE;
				fbMBRead_FC3.bExecute := FALSE;
					iSFPowerMPPT := 0;
						wNumberOfMPPT := 0;
							wNextModbusStartAdress := 0;
								wNumberOfInputs := 0;
									lrRestNextAdress := 0;	
	
		//Set Firmer Output Structure to default
		stFirmerInverterData.rTotalMPPTPower := 0;
			stFirmerInverterData.rCabinetTemp := 0;
				stFirmerInverterData.rHeatSinkTemp := 0;
					FOR byLPFillDefaultData := 1 TO 6 BY 1 DO
						stFirmerInverterData.arrMPPTPower[byLPFillDefaultData] := 0;
					END_FOR
						stFirmerInverterData.eEvent1 := eFirmerEvent.eNoInfo;
							stFirmerInverterData.eOperatingState := eFirmerOperatingState.eNoInfo;
								stFirmerInverterData.eVendorEvent1 := eFirmerVendorEvent1.eNoInfo;
									stFirmerInverterData.eVendorEvent2 := eFirmerVendorEvent2.eNoInfo;
										stFirmerInverterData.eVendorEvent3 := eFirmerVendorEvent3.eNoInfo;	
	
	1://Read Out Values from Pic 103 of the Sunspec Protocol (Register 40073)
		iStateModbus_CP := iStateModbusRead;
		
		//Start Read
		fbMBRead_FC3.nQuantity := 45;
			fbMBRead_FC3.nMBAddr := 40073;
				fbMBRead_FC3.bExecute := TRUE;
					fbMBRead_FC3.nUnitID := byUnitID_Inverter;
		
		IF fbMBRead_FC3.bBusy THEN timDelay.IN := TRUE; END_IF

		//Copy the read out Data
		IF NOT fbMBRead_FC3.bBusy AND NOT fbMBRead_FC3.bError AND timDelay.Q THEN
			//Current L1
			IF WORD_TO_INT(arrBuffer_FC3[4]) >= - 10 AND WORD_TO_INT(arrBuffer_FC3[4]) <= 10 THEN
				fbElMeter.lrCurrentL1 := arrBuffer_FC3[1] * EXPT(10,WORD_TO_INT(arrBuffer_FC3[4]));
			END_IF
			//Current L2
			IF WORD_TO_INT(arrBuffer_FC3[4]) >= - 10 AND WORD_TO_INT(arrBuffer_FC3[4]) <= 10 THEN
				fbElMeter.lrCurrentL2 := arrBuffer_FC3[2] * EXPT(10,WORD_TO_INT(arrBuffer_FC3[4]));
			END_IF
			//Current L3
			IF WORD_TO_INT(arrBuffer_FC3[4]) >= - 10 AND WORD_TO_INT(arrBuffer_FC3[4]) <= 10 THEN
				fbElMeter.lrCurrentL3 := arrBuffer_FC3[3] * EXPT(10,WORD_TO_INT(arrBuffer_FC3[4]));
			END_IF
			//Voltage L1/N
			IF WORD_TO_INT(arrBuffer_FC3[11]) >= - 10 AND WORD_TO_INT(arrBuffer_FC3[11]) <= 10 THEN
				fbElMeter.lrVoltageL1N := arrBuffer_FC3[8] * EXPT(10,WORD_TO_INT(arrBuffer_FC3[11]));
			END_IF
			//Voltage L2/N
			IF WORD_TO_INT(arrBuffer_FC3[11]) >= - 10 AND WORD_TO_INT(arrBuffer_FC3[11]) <= 10 THEN
				fbElMeter.lrVoltageL2N := arrBuffer_FC3[9] * EXPT(10,WORD_TO_INT(arrBuffer_FC3[11]));
			END_IF
			//Voltage L3/N
			IF WORD_TO_INT(arrBuffer_FC3[11]) >= - 10 AND WORD_TO_INT(arrBuffer_FC3[11]) <= 10 THEN
				fbElMeter.lrVoltageL3N := arrBuffer_FC3[10] * EXPT(10,WORD_TO_INT(arrBuffer_FC3[11]));
			END_IF
			//AC Power
			IF WORD_TO_INT(arrBuffer_FC3[13]) >= - 10 AND WORD_TO_INT(arrBuffer_FC3[13]) <= 10 THEN  
				fbElMeter.lrPowerTotal := WORD_TO_INT(arrBuffer_FC3[12]) * EXPT(10,WORD_TO_INT(arrBuffer_FC3[13]));
			END_IF
			//Hz
			IF WORD_TO_INT(arrBuffer_FC3[15]) >= - 10 AND WORD_TO_INT(arrBuffer_FC3[15]) <= 10 THEN  
				fbElMeter.lrFrequency := arrBuffer_FC3[14] * EXPT(10,WORD_TO_INT(arrBuffer_FC3[15]));
			END_IF
			//Apparent Power
			IF WORD_TO_INT(arrBuffer_FC3[17]) >= - 10 AND WORD_TO_INT(arrBuffer_FC3[17]) <= 10 THEN  
				fbElMeter.lrApparentPowerTotal := WORD_TO_INT(arrBuffer_FC3[16]) * EXPT(10,WORD_TO_INT(arrBuffer_FC3[17]));
			END_IF
			//Reactive Power
			IF WORD_TO_INT(arrBuffer_FC3[19]) >= - 10 AND WORD_TO_INT(arrBuffer_FC3[19]) <= 10 THEN  
				fbElMeter.lrReactivePowerTotal := WORD_TO_INT(arrBuffer_FC3[18]) * EXPT(10,WORD_TO_INT(arrBuffer_FC3[19]));
			END_IF
			//Produced Energy
			IF WORD_TO_INT(arrBuffer_FC3[24]) >= - 10 AND WORD_TO_INT(arrBuffer_FC3[24]) <= 10 THEN  
				fbConvertWord(wInputValue_1:= arrBuffer_FC3[22], wInputValue_2:= arrBuffer_FC3[23], eByteOrderForConvert:= eByteOrder.eBigEndian, dwOutputValue=> );
					fbElMeter.lrCounterEnergyT1_Production := fbConvertWord.dwOutputValue * EXPT(10,WORD_TO_INT(arrBuffer_FC3[24]));
						fbElMeter.lrCounterEnergyT1_Production := fbElMeter.lrCounterEnergyT1_Production / 1000;
							fbElMeter.lrTotalCounterEnergy_Production := fbElMeter.lrCounterEnergyT1_Production; 	
			END_IF
			//Cabinet Temperature
			IF WORD_TO_INT(arrBuffer_FC3[35]) >= - 10 AND WORD_TO_INT(arrBuffer_FC3[35]) <= 10 THEN  
				stFirmerInverterData.rCabinetTemp := LREAL_TO_REAL(WORD_TO_INT(arrBuffer_FC3[31]) * EXPT(10,WORD_TO_INT(arrBuffer_FC3[35])));
			END_IF
			//Heat Sink Temperature
			IF WORD_TO_INT(arrBuffer_FC3[35]) >= - 10 AND WORD_TO_INT(arrBuffer_FC3[35]) <= 10 THEN  
				stFirmerInverterData.rHeatSinkTemp := LREAL_TO_REAL(WORD_TO_INT(arrBuffer_FC3[32]) * EXPT(10,WORD_TO_INT(arrBuffer_FC3[35])));
			END_IF
			//Operating State
			stFirmerInverterData.eOperatingState := eFirmerOperatingState.eNoInfo;
			IF arrBuffer_FC3[36] = 1 THEN stFirmerInverterData.eOperatingState := eFirmerOperatingState.eOff;
			ELSIF arrBuffer_FC3[36] = 2 THEN stFirmerInverterData.eOperatingState := eFirmerOperatingState.eSleeping;
			ELSIF arrBuffer_FC3[36] = 3 THEN stFirmerInverterData.eOperatingState := eFirmerOperatingState.eStarting;
			ELSIF arrBuffer_FC3[36] = 4 THEN stFirmerInverterData.eOperatingState := eFirmerOperatingState.eMppt;
			ELSIF arrBuffer_FC3[36] = 5 THEN stFirmerInverterData.eOperatingState := eFirmerOperatingState.eThrottled;
			ELSIF arrBuffer_FC3[36] = 6 THEN stFirmerInverterData.eOperatingState := eFirmerOperatingState.eShuttingDown;
			ELSIF arrBuffer_FC3[36] = 7 THEN stFirmerInverterData.eOperatingState := eFirmerOperatingState.eFault;
			ELSIF arrBuffer_FC3[36] = 8 THEN stFirmerInverterData.eOperatingState := eFirmerOperatingState.eStandby;
			END_IF 
			//Event 1
			fbConvertWord(wInputValue_1:= arrBuffer_FC3[38], wInputValue_2:= arrBuffer_FC3[39], eByteOrderForConvert:= eByteOrder.eBigEndian, dwOutputValue=> );
			stFirmerInverterData.eEvent1 := eFirmerEvent.eNoInfo;
			IF fbConvertWord.dwOutputValue.0 THEN stFirmerInverterData.eEvent1 := eFirmerEvent.eGroundFault;
			ELSIF fbConvertWord.dwOutputValue.1 THEN stFirmerInverterData.eEvent1 := eFirmerEvent.eDCOverVolt;
			ELSIF fbConvertWord.dwOutputValue.2 THEN stFirmerInverterData.eEvent1 := eFirmerEvent.eACDisconnect;
			ELSIF fbConvertWord.dwOutputValue.3 THEN stFirmerInverterData.eEvent1 := eFirmerEvent.eDCDisconnect;
			ELSIF fbConvertWord.dwOutputValue.4 THEN stFirmerInverterData.eEvent1 := eFirmerEvent.eGridDisconnect;
			ELSIF fbConvertWord.dwOutputValue.5 THEN stFirmerInverterData.eEvent1 := eFirmerEvent.eCabinetOpen;
			ELSIF fbConvertWord.dwOutputValue.6 THEN stFirmerInverterData.eEvent1 := eFirmerEvent.eManualShutdown;
			ELSIF fbConvertWord.dwOutputValue.7 THEN stFirmerInverterData.eEvent1 := eFirmerEvent.eOverTemp;
			ELSIF fbConvertWord.dwOutputValue.8 THEN stFirmerInverterData.eEvent1 := eFirmerEvent.eOverFrequency;
			ELSIF fbConvertWord.dwOutputValue.9 THEN stFirmerInverterData.eEvent1 := eFirmerEvent.eUnderFrequency;
			ELSIF fbConvertWord.dwOutputValue.10 THEN stFirmerInverterData.eEvent1 := eFirmerEvent.eACOverVolt;
			ELSIF fbConvertWord.dwOutputValue.11 THEN stFirmerInverterData.eEvent1 := eFirmerEvent.eACUnderVolt;
			ELSIF fbConvertWord.dwOutputValue.12 THEN stFirmerInverterData.eEvent1 := eFirmerEvent.eBlownStringFuse;
			ELSIF fbConvertWord.dwOutputValue.13 THEN stFirmerInverterData.eEvent1 := eFirmerEvent.eUnderTemp;
			ELSIF fbConvertWord.dwOutputValue.14 THEN stFirmerInverterData.eEvent1 := eFirmerEvent.eMemoryLoss;
			ELSIF fbConvertWord.dwOutputValue.15 THEN stFirmerInverterData.eEvent1 := eFirmerEvent.eHWTestFailure;
			END_IF
			//Vendor Event 1
			fbConvertWord(wInputValue_1:= arrBuffer_FC3[40], wInputValue_2:= arrBuffer_FC3[41], eByteOrderForConvert:= eByteOrder.eBigEndian, dwOutputValue=> );
			stFirmerInverterData.eVendorEvent1 := eFirmerVendorEvent1.eNoInfo;
			IF fbConvertWord.dwOutputValue.0 THEN stFirmerInverterData.eVendorEvent1 := eFirmerVendorEvent1.ePowerCurtailmentFromExternalCommand;
			ELSIF fbConvertWord.dwOutputValue.1 THEN stFirmerInverterData.eVendorEvent1 := eFirmerVendorEvent1.ePowerLimitationFromFrequencyWatt;
			ELSIF fbConvertWord.dwOutputValue.2 THEN stFirmerInverterData.eVendorEvent1 := eFirmerVendorEvent1.ePowerLimitationFromHighAverageGridVoltage;
			ELSIF fbConvertWord.dwOutputValue.3 THEN stFirmerInverterData.eVendorEvent1 := eFirmerVendorEvent1.ePowerLimitationFromAntiIslandingProtection;
			ELSIF fbConvertWord.dwOutputValue.4 THEN stFirmerInverterData.eVendorEvent1 := eFirmerVendorEvent1.ePowerLimitationFromGridCurrentRatingLimitation;
			ELSIF fbConvertWord.dwOutputValue.5 THEN stFirmerInverterData.eVendorEvent1 := eFirmerVendorEvent1.ePowerLimitationForHighTemperature;
			ELSIF fbConvertWord.dwOutputValue.6 THEN stFirmerInverterData.eVendorEvent1 := eFirmerVendorEvent1.ePowerLimitationForHighDCVoltage;
			ELSIF fbConvertWord.dwOutputValue.8 THEN stFirmerInverterData.eVendorEvent1 := eFirmerVendorEvent1.ePowerLimitationFromRampRateConnectionRamp;
			ELSIF fbConvertWord.dwOutputValue.9 THEN stFirmerInverterData.eVendorEvent1 := eFirmerVendorEvent1.ePowerLimitationFromMomentaryCessation;
			ELSIF fbConvertWord.dwOutputValue.10 THEN stFirmerInverterData.eVendorEvent1 := eFirmerVendorEvent1.ePowerLimitationFromRampRateNormalRampUp;
			ELSIF fbConvertWord.dwOutputValue.11 THEN stFirmerInverterData.eVendorEvent1 := eFirmerVendorEvent1.ePowerLimitationFromVoltWatt;
			ELSIF fbConvertWord.dwOutputValue.12 THEN stFirmerInverterData.eVendorEvent1 := eFirmerVendorEvent1.ePowerLimitationFromCapabilityRating;	
			END_IF
			//Vendor Event 2
			fbConvertWord(wInputValue_1:= arrBuffer_FC3[42], wInputValue_2:= arrBuffer_FC3[43], eByteOrderForConvert:= eByteOrder.eBigEndian, dwOutputValue=> );
			stFirmerInverterData.eVendorEvent2 := eFirmerVendorEvent2.eNoInfo;
			IF fbConvertWord.dwOutputValue.0 THEN stFirmerInverterData.eVendorEvent2 := eFirmerVendorEvent2.ePowerLimitationForHighTemperature;
			ELSIF fbConvertWord.dwOutputValue.1 THEN stFirmerInverterData.eVendorEvent2 := eFirmerVendorEvent2.ePowerLimitationForHighDCVoltage;
			ELSIF fbConvertWord.dwOutputValue.2 THEN stFirmerInverterData.eVendorEvent2 := eFirmerVendorEvent2.ePowerLimitationFromCapabilityRating;	
			END_IF
			//Vendor Event 3
			fbConvertWord(wInputValue_1:= arrBuffer_FC3[44], wInputValue_2:= arrBuffer_FC3[45], eByteOrderForConvert:= eByteOrder.eBigEndian, dwOutputValue=> );
			stFirmerInverterData.eVendorEvent3 := eFirmerVendorEvent3.eNoInfo;
			IF fbConvertWord.dwOutputValue.0 THEN stFirmerInverterData.eVendorEvent3 := eFirmerVendorEvent3.eFanFault;
			ELSIF fbConvertWord.dwOutputValue.1 THEN stFirmerInverterData.eVendorEvent3 := eFirmerVendorEvent3.eStatisticsMemoryFault;
			ELSIF fbConvertWord.dwOutputValue.2 THEN stFirmerInverterData.eVendorEvent3 := eFirmerVendorEvent3.eRTCClockNotSet;
			ELSIF fbConvertWord.dwOutputValue.4 THEN stFirmerInverterData.eVendorEvent3 := eFirmerVendorEvent3.eRTCLowBatteryFault;
			ELSIF fbConvertWord.dwOutputValue.5 THEN stFirmerInverterData.eVendorEvent3 := eFirmerVendorEvent3.eRTCQuartzFault;	
			END_IF
			
			//Go to Next Step
			fbMBRead_FC3.bExecute := FALSE;
				timDelay.IN := FALSE;		
					iStateModbusRead := 2;	
						wNextModbusStartAdress := 40122;
		END_IF

		//Error or Timeout
		IF FPError_FC_3.Q OR timTimeout.Q THEN
			iStateModbusError := 300;
		END_IF
	
	2://Read Out Values from Pic 120 to Start Adress for PIC 160 of the Sunspec Protocoll		
		iStateModbus_CP := iStateModbusRead;
		
		//Start Read
		fbMBRead_FC3.nQuantity := 2;
			fbMBRead_FC3.nMBAddr := wNextModbusStartAdress;
				fbMBRead_FC3.bExecute := TRUE;
					fbMBRead_FC3.nUnitID := byUnitID_Inverter;
		
		IF fbMBRead_FC3.bBusy THEN timDelay.IN := TRUE; END_IF

		//Copy the read out Data
		IF NOT fbMBRead_FC3.bBusy AND NOT fbMBRead_FC3.bError AND timDelay.Q THEN
			//PIC ID
			wPicID := arrBuffer_FC3[1];
			//Number of Inputs
			wNumberOfInputs := arrBuffer_FC3[2];
			
			//Go to Next Step
			fbMBRead_FC3.bExecute := FALSE;
				timDelay.IN := FALSE;		
					iStateModbusRead := 3;	
						lrRestNextAdress := 0;
							//Calculate next Modbus Start Adress for next Pic
							wNextModbusStartAdress := wNextModbusStartAdress + wNumberOfInputs + 2;
								lrRestNextAdress := FRAC(WORD_TO_REAL(wNextModbusStartAdress) / 2);	
									//If it ends with an odd number, the next PIC starts with an even address
									IF lrRestNextAdress <> 0 THEN wNextModbusStartAdress := wNextModbusStartAdress + 1; END_IF
		END_IF     					
		
		//Error or Timeout
		IF FPError_FC_3.Q OR timTimeout.Q THEN
			iStateModbusError := 300;
		END_IF	
	
	3://Check the PIC ID
		iStateModbus_CP := iStateModbusRead;
		
		IF wPicID < 160 THEN
			//Back to Step 2
			iStateModbusRead := 2;
		ELSE
			//next Step with values
			iStateModbusRead := 4;
				//Calculate next Modbus Start Adress for next Pic
				wNextModbusStartAdress := wNextModbusStartAdress - wNumberOfInputs - 2;
		END_IF
		
	
	4://Read Out Values from Pic 160 of the Sunspec Protocol
		iStateModbus_CP := iStateModbusRead;
		
		//Start Read
		fbMBRead_FC3.nQuantity := 9;
			fbMBRead_FC3.nMBAddr := wNextModbusStartAdress;
				fbMBRead_FC3.bExecute := TRUE;
					fbMBRead_FC3.nUnitID := byUnitID_Inverter;
		
		IF fbMBRead_FC3.bBusy THEN timDelay.IN := TRUE; END_IF

		//Copy the read out Data
		IF NOT fbMBRead_FC3.bBusy AND NOT fbMBRead_FC3.bError AND timDelay.Q THEN
			//PIC ID
			wPicID := arrBuffer_FC3[1];
			//Number of Inputs
			wNumberOfInputs := arrBuffer_FC3[2];
			//Scale Factor for String Power
			iSFPowerMPPT := WORD_TO_INT(arrBuffer_FC3[5]);
			//Number of MPPT Moduls
			wNumberOfMPPT := arrBuffer_FC3[9];
			
			//Go to Next Step
			fbMBRead_FC3.bExecute := FALSE;
				timDelay.IN := FALSE;		
					iStateModbusRead := 5;	
						wNextModbusStartAdress := wNextModbusStartAdress + 10;
		END_IF     				
		
		//Error or Timeout
		IF FPError_FC_3.Q OR timTimeout.Q THEN
			iStateModbusError := 300;
		END_IF

	5://Read Out Values from Pic 160 of the Sunspec Protocol
		iStateModbus_CP := iStateModbusRead;
		
		//Start Read
		fbMBRead_FC3.nQuantity := 20 * wNumberOfMPPT;
			fbMBRead_FC3.nMBAddr := wNextModbusStartAdress;
				fbMBRead_FC3.bExecute := TRUE;
					fbMBRead_FC3.nUnitID := byUnitID_Inverter;
		
		wNumberOfMPPT := LIMIT(1,wNumberOfMPPT,6);
			iSFPowerMPPT := LIMIT(-10,iSFPowerMPPT,10);
		
		IF fbMBRead_FC3.bBusy THEN timDelay.IN := TRUE; END_IF

		IF wNumberOfMPPT <= 1 THEN
			stFirmerInverterData.arrMPPTPower[2] := 0;
				stFirmerInverterData.arrMPPTPower[3] := 0;
					stFirmerInverterData.arrMPPTPower[4] := 0;
						stFirmerInverterData.arrMPPTPower[5] := 0;
							stFirmerInverterData.arrMPPTPower[6] := 0;
		ELSIF  wNumberOfMPPT = 2 THEN
			stFirmerInverterData.arrMPPTPower[3] := 0;
				stFirmerInverterData.arrMPPTPower[4] := 0;
					stFirmerInverterData.arrMPPTPower[5] := 0;
						stFirmerInverterData.arrMPPTPower[6] := 0;
		ELSIF  wNumberOfMPPT = 3 THEN
			stFirmerInverterData.arrMPPTPower[4] := 0;
				stFirmerInverterData.arrMPPTPower[5] := 0;
					stFirmerInverterData.arrMPPTPower[6] := 0;
		ELSIF  wNumberOfMPPT = 4 THEN
			stFirmerInverterData.arrMPPTPower[5] := 0;
				stFirmerInverterData.arrMPPTPower[6] := 0;	
		ELSIF  wNumberOfMPPT = 5 THEN
			stFirmerInverterData.arrMPPTPower[6] := 0;
		END_IF
		
		//Copy the read out Data
		IF NOT fbMBRead_FC3.bBusy AND NOT fbMBRead_FC3.bError AND timDelay.Q THEN
			//MPPT Power
			FOR wLPPowerMPPT := 1 TO (20 * wNumberOfMPPT) BY 1 DO
				IF wNumberOfMPPT >= 1 AND wLPPowerMPPT = 12 THEN stFirmerInverterData.arrMPPTPower[1] := LREAL_TO_REAL(arrBuffer_FC3[wLPPowerMPPT] * EXPT(10,iSFPowerMPPT) / 1000);
				ELSIF wNumberOfMPPT >= 2 AND wLPPowerMPPT = 32 THEN stFirmerInverterData.arrMPPTPower[2] := LREAL_TO_REAL(arrBuffer_FC3[wLPPowerMPPT] * EXPT(10,iSFPowerMPPT) / 1000);
				ELSIF wNumberOfMPPT >= 3 AND wLPPowerMPPT = 52 THEN stFirmerInverterData.arrMPPTPower[3] := LREAL_TO_REAL(arrBuffer_FC3[wLPPowerMPPT] * EXPT(10,iSFPowerMPPT) / 1000);
				ELSIF wNumberOfMPPT >= 4 AND wLPPowerMPPT = 72 THEN stFirmerInverterData.arrMPPTPower[4] := LREAL_TO_REAL(arrBuffer_FC3[wLPPowerMPPT] * EXPT(10,iSFPowerMPPT) / 1000);
				ELSIF wNumberOfMPPT >= 5 AND wLPPowerMPPT = 92 THEN stFirmerInverterData.arrMPPTPower[5] := LREAL_TO_REAL(arrBuffer_FC3[wLPPowerMPPT] * EXPT(10,iSFPowerMPPT) / 1000);
				ELSIF wNumberOfMPPT >= 6 AND wLPPowerMPPT = 112 THEN stFirmerInverterData.arrMPPTPower[6] := LREAL_TO_REAL(arrBuffer_FC3[wLPPowerMPPT] * EXPT(10,iSFPowerMPPT) / 1000);
				END_IF     
			END_FOR 
			
			//Go to Next Step
			fbMBRead_FC3.bExecute := FALSE;
				timDelay.IN := FALSE;		
					iStateModbusRead := 1;
						byErrorCounterTCP := 0;
							iSFPowerMPPT := 0;
								wNumberOfMPPT := 0;
									wNextModbusStartAdress := 0;
										wNumberOfInputs := 0;
											lrRestNextAdress := 0;
		END_IF     				
		
		//Total DC Power
		stFirmerInverterData.rTotalMPPTPower := 0;
			FOR wLPPowerMPPT := 1 TO 6 BY 1 DO
				stFirmerInverterData.rTotalMPPTPower := stFirmerInverterData.rTotalMPPTPower + stFirmerInverterData.arrMPPTPower[wLPPowerMPPT];
			END_FOR
			
		//Error or Timeout
		IF FPError_FC_3.Q OR timTimeout.Q THEN
			iStateModbusError := 300;
		END_IF
	
END_CASE

(*------------------------------------------------------------------Error and Warning----------------------------------------------------------------------------*)	

bErrorInverter := FALSE;
	IF stFirmerInverterData.eOperatingState = eFirmerOperatingState.eFault THEN bErrorInverter := TRUE; END_IF
		IF stFirmerInverterData.eEvent1 <> eFirmerEvent.eNoInfo THEN bErrorInverter := TRUE; END_IF
			IF stFirmerInverterData.eVendorEvent3 <> eFirmerVendorEvent3.eNoInfo THEN bErrorInverter := TRUE; END_IF     

IF timDissableFunctions.Q OR stFirmerInverterData.eVendorEvent1 <> eFirmerVendorEvent1.eNoInfo OR stFirmerInverterData.eVendorEvent2 <> eFirmerVendorEvent2.eNoInfo THEN fbElMeter.bWarning := TRUE; ELSE fbElMeter.bWarning := FALSE; fbElMeter.iWarningCode := 0; END_IF   
	IF Lynus_Standards.GVL_Energy.stNumberOfDevices.diNumberOfElectricMeters > Constants_Energy.diMaxNumberOfElectricMeters OR bErrorInverter OR byErrorCounterTCP > 10 THEN 
		fbElMeter.bError := TRUE;
	ELSE 
		fbElMeter.bError := FALSE;
			fbElMeter.iErrorCode := 0;
	END_IF

IF stFirmerInverterData.eVendorEvent1 <> eFirmerVendorEvent1.eNoInfo OR stFirmerInverterData.eVendorEvent2 <> eFirmerVendorEvent2.eNoInfo THEN fbElMeter.iWarningCode := 1; END_IF   	
	
IF Lynus_Standards.GVL_Energy.stNumberOfDevices.diNumberOfElectricMeters > Constants_Energy.diMaxNumberOfElectricMeters THEN fbElMeter.iErrorCode := 1; END_IF
	IF byErrorCounterTCP > 10 OR bErrorInverter THEN fbElMeter.iErrorCode := 0; END_IF   

(*------------------------------------------------------------------Logic----------------------------------------------------------------------------*)

//Read Out Data done for EM Function
IF iStateModbusRead <> 1 THEN fbElMeter.bReadOutDataDone := TRUE; ELSE fbElMeter.bReadOutDataDone := FALSE; END_IF

//Function block for meter data
fbElMeter(
	bEnable:= bEnable AND NOT timDissableFunctions.Q, 
	bError:= , 
	bEnableReadOutFunction:= FALSE, 
	bWriteWithDelay:= TRUE,
	bPowerDataInvers:= FALSE, 
	bReadOutDataDone:= ,
	iTimeReadOutInterval:= , 
	iErrorCode:= , 
	iWarningCode:= , 
	lrTotalCounterEnergy_Consumption:= 0, 
	lrTotalCounterEnergy_Production:= , 
	lrCounterEnergyT1_Consumption:= 0, 
	lrCounterEnergyT2_Consumption:= 0, 
	lrCounterEnergyT1_Production:= , 
	lrCounterEnergyT2_Production:= 0, 
	lrCurrentL1:= , 
	lrVoltageL1N:= , 
	lrVoltageL1L2:= , 
	lrPowerL1:= 0, 
	lrCurrentL2:= , 
	lrVoltageL2N:= , 
	lrVoltageL2L3:= , 
	lrPowerL2:= 0, 
	lrCurrentL3:= , 
	lrVoltageL3N:= , 
	lrVoltageL3L1:= , 
	lrPowerL3:= 0, 
	lrPowerTotal:= , 
	lrFrequency:= , 
	lrReactivePowerTotal:= , 
	lrApparentPowerTotal:= , 
	tTimDelayOutput:= T#5S, 
	stDataEMOutPower=> , 
	stDataEMOutPowerDelay=> stDataEMPower_PV, 
	stDataEMOutCounter=> ,
	stDataEMOutCounterDelay=> stDataEMCounter_PV, 
	bReadOutMeter=> );
	
(*------------------------------------------------------------------------------------------State Machine Error---------------------------------------------------------------------------------------------*)	

CASE iStateModbusError OF
	
	300://Error
		iStateModbus_CP := iStateModbusError;
			timDelay.IN := FALSE;
				fbMBRead_FC3.bExecute := FALSE;
					iSFPowerMPPT := 0;
						wNumberOfMPPT := 0;
							wNextModbusStartAdress := 0;
								wNumberOfInputs := 0;
									lrRestNextAdress := 0;
										byErrorCounterTCP := byErrorCounterTCP + 1;
										byErrorCounterTCP := LIMIT(0,byErrorCounterTCP,11);
											//Restart from new with the Read out part after an Error
											IF byErrorCounterTCP < 10 THEN
												iStateModbusRead := 1;
													iStateModbusError := 0;
											ELSE
												//Wait here in the Error State for the Delay Timer and then we dont have a Timeout Error
												iStateModbusRead := - 1;
													//Start from New when the Delay is paste
													IF timCloseSocket.Q THEN
														iStateModbusRead := 1;	
															iStateModbusError := 0;
																byErrorCounterTCP := 0;
													END_IF	
											END_IF
END_CASE

//Timer to close the Socket after to much TCP Errors and reopen a new one
timCloseSocket(IN:= byErrorCounterTCP > 10 AND fbElMeter.stDataEMOutPower.bEnabled, PT:= T#1M, Q=> , ET=> );

(*------------------------------------------------------------------------------------------Modbus TCP Function---------------------------------------------------------------------------------------------*)

fbMBRead_FC3(sIPAddr:= sIPAdress, nTCPPort:= 502, cbLength:= SIZEOF(arrBuffer_FC3), pDestAddr:= ADR(arrBuffer_FC3), tTimeout:= T#10S );
	FPError_FC_3(CLK:= fbMBRead_FC3.bError, Q=> );

(*-----------------------------------------------------------Handle data to Global structure for Electric Meter system and Modbus RTU Communication-----------------------------------------------------------------*)

CASE iStateGVLData OF
	
	0://Init Step
		byWaitInStep := 0;
			diCounterForGVL := 1;
	
	1://Wait for 4 Steps before clean al Data on GVL
		byWaitInStep := byWaitInStep + 1;
			IF byWaitInStep >= 4 AND fbNumberDevice.bNumberIsCalculatet THEN iStateGVLData := 2; END_IF
				//To much Devices, back to the Init step
				IF byWaitInStep >= 4 AND NOT fbNumberDevice.bNumberIsCalculatet THEN iStateGVLData := 0; END_IF	
			
